# B&R Automation Studio project TD52 (part 107)

#### ERDFCyclic.st - Cyclic code
```iecst
(*********************************************************************************************
AGGR: ERDF task (cyclic)

This code is confidential AND proprietary to the INNIO Company.
It may NOT be used in any form, or reproduced in any manner, without the express
written permission of the INNIO Company.
Copyright, INNIO Company, 2019

Customized modifications: -
------------------------

History:
-------
 V0.1:  Kirchler 02.05.2012: Anwahl Leistungsvorgabe durch ERDF aucb wenn Sollwert über BUS
 							 Signal Aggregat nicht verfügbar wird nicht gesetzt wenn A_ANF fehlt
 V0.2:  Kirchler 17.07.2012: Komplett umgebaut laut vorgabe Clarke; Alle eingänge auf Impuls/flankenauswertung
 							 Leistungsvorgabe und Blindleistungsvorgabe als Reduktion (maximum)
							 RSE Signal implementiert
 V0.3:	Kirchler 13.09.2012: ERDF Schnittstellen aktiv auch im Handbetrieb
 							 Merken der aktuell ausgewählten Cosphi Funktion und nach Beendigung Q0 LIMIT wieder auf alten Wert stellen
							 Vereinfachungen Teil P0- und Q0-Limitierungen
 V0.4:  Kirchler 25.10.2012: Q0 Limitierung Set nur möglich wenn Q0 inaktiv und Reset nur möglich wenn Q0 aktiv.
 							 Verhindert QPF Funktions-Parameter Überschreibungen
							 Wenn Q0_max grösser aktuelle Blindleistung einfach auf alten Cosphi modus zurückschalten
 V0.5:  Adami 07.11.2012: 	 Fehler behoben mit der Netzstörung >50 Sek und der Entkopplung vom netz durch DEIE. Die 2 Funktionen blockierten sich gegenseitig, dadurch
 							 konnte man keine der beiden mehr resetten und die Maschine nicht mehr starten	(außer durch einen Neustart der Diane)
 							 Funktionsänderung der Variablen "DO_NotReady ". Dieser Ausgang dient jetzt als "watchdog", d.h der Ausgang soll immer "1" sein sobald die SPS läuft.
							 Anpassung Blindleistungsreduzierung
 V0.6   Kirchmair 06.02.2014:Erestzen der Variable DI_EVU_3 durch DI_EVU_BLOCK, da sich die Funktion der Variable DI_EVU_3 geändert hat (seit V3.4) und jetzt nicht mehr verwendbar ist.

 V4.00.0 28-04-2014 Maxhera/Waldhart,   implementation OF the module FOR modular software
 V4.03.0 15-03-2016	Perktold,	update FOR 4.3.0.0
 V4.04.0 06-10-2016	Perktold,	update FOR 4.4.0.0 (tiDelayDEIE, IN_GR.tPLim_DEIE.Ai)
		 09.10.2019	lettenb.	div.by zero bugfix, bu01

Instructions FOR use:
--------------------
-
Outstandings:
-------------
*********************************************************************************************)

PROGRAM _CYCLIC

IF Para.bDEIE_Active THEN
(* requirement coupling / decoupling from EU (ERDF), Digital inputs *)
	xSR_MCB_Dcp(SET1 := IN_GR.tMCB_Dcp_SetEUCOn.Di, RESET := IN_GR.tMCB_Dcp_SetEUCOf.Di);
	bMCB_Dcp		 := xSR_MCB_Dcp.Q1;

(* feedback Receive requested Command form machine*)
	IF bMCB_Dcp THEN 						(* True --> hier wird der motor abgefordert *)
		OUT_GR.tMCB_SOn.Do 		:= TRUE;	(* rückmeldung für abforderung *)
		OUT_GR.tERDF_BLOCK.Do 	:= TRUE;   	(* TRUE = abforderung des Motors *)
 	ELSE									(* motor ist wieder freigegeben *)
		OUT_GR.tMCB_SOn.Do		:= FALSE;
		OUT_GR.tERDF_BLOCK.Do 	:= FALSE; 	(* FALSE = keine abforderung des motors durch erdf  *)
	END_IF;

(* =====================================================================*)

(* Freigabe Kopplung ans Netz durch ERDF / Release coupling to the grid by ERDF *)
	xTON_GTE(IN :=  NOT IN_GR.tMnsOk_GTE.Di, PT := Para.tiDelayDEIE);   (* network trouble after X[s]  *)
	xSR_MCB_RelSync(SET1 := IN_GR.tMCB_Rel_Sync.Di, RESET := xTON_GTE.Q);
	bMCB_RelSync := xSR_MCB_RelSync.Q1; (* FALSE = Motor soll blockieren *)

	TP_Msg2888(IN := bMCB_RelSync, PT := T#15s);
	bMsg2888	:= TP_Msg2888.Q;

	IF bMCB_RelSync THEN		(* True --> freigabe für sy erteilt --> keine blockierung *)
		OUT_GR.bOpAlm_ERDF_SY	:= OUT_GR.tMCB_Rel_Sync_SOn.Do := TRUE;	(* rückmeldung und betiebsmeldung abgesetzt *)
	ELSE
		OUT_GR.bOpAlm_ERDF_SY	:= OUT_GR.tMCB_Rel_Sync_SOn.Do := FALSE;
	END_IF;
(* =====================================================================*)

(*  DO: Generator ist eingeschaltet / Generator switch is on *)
	OUT_GR.tGCB_SOn.Do 			:= IN_GR.tGCB_On.Di;
(* =====================================================================*)

(* Fast decoupled by ERDF / Schnelles entkoppeln durch ERDF	*)
(* requirement coupling / decoupling quickly from EU (ERDF), Digital inputs *)
	xSR_MCB_DcpQu(SET1 := IN_GR.tMCB_DcpQu_SetEUCOn.Di, RESET := IN_GR.tMCB_DcpQu_SetEUCOf.Di);
	bMCB_DcpQu	  := xSR_MCB_DcpQu.Q1;

	IF bMCB_DcpQu THEN
		OUT_GR.bOpAlm_DecQu 	:= TRUE;
		OUT_GR.tMCB_EDF_SOn.Do	:= TRUE;
	ELSE
		OUT_GR.bOpAlm_DecQu 	:= FALSE;
		OUT_GR.tMCB_EDF_SOn.Do	:= FALSE;
	END_IF;
(* =====================================================================*)

(*Customers switch for bridging P0 signal / Kundenschalter zur Überbrückung P0 Signal*)
	IF IN_GR.tP0_BLOCK_DEIE.Di THEN
		IN_GR.tPLim_GenC_SetEU.Ai 	:= Para.rP_Set_ExtAI_NormScalMax;
	ELSE
		IN_GR.tPLim_GenC_SetEU.Ai  	:= IN_GR.tP_DEIE.Ai;
	END_IF;

	IF bGCP_PLim AND NOT IN_GR.tP0_BLOCK_DEIE.Di THEN
		OUT_GR.bOpMsg_Plim_ERDF_SOnOf	:= TRUE;
	END_IF;

	IF NOT bGCP_PLim OR  IN_GR.tP0_BLOCK_DEIE.Di THEN
		OUT_GR.bOpMsg_Plim_ERDF_SOnOf	:= FALSE;
	END_IF;

(* powerlimit from ERDF / Leistung reduktion von ERDF *)
	IF  OUT_GR.tPLim_GenC_SOn.Do AND  (IN_GR.tPLim_GenC_SetEU.Ai< (IN_GR.rP_Nom * 0.5)) THEN	(* abforderung des motors sollte die leistungsreduktion < 50% sein *)
		OUT_GR.bOpMsg_Plim_ERDF_ABF_SOnOf	:= TRUE;		(* true = abforderung des Motors *)
	ELSE
		OUT_GR.bOpMsg_Plim_ERDF_ABF_SOnOf 	:= FALSE;
		IN_GR.tPLim_GenC_SetEU.Ai	  		:= LIMIT ((IN_GR.rP_Nom * 0.5), IN_GR.tPLim_GenC_SetEU.Ai,IN_GR.rP_Nom);
		rP_Red_ERDF_Lim			 	  		:= IN_GR.tPLim_GenC_SetEU.Ai / MAX(1, IN_GR.rP_Nom);
	END_IF;
	IF NOT OUT_GR.tPLim_GenC_SOn.Do THEN					(* no powerlimit from ERDF / keine Leistung reduktion über ERDF *)
		rP_Red_ERDF_Lim						:= 1.0; 		(* maximum power / maximale Leistung *)
		OUT_GR.bOpMsg_Plim_ERDF_SOnOf  		:= FALSE;
	END_IF;

(* =====================================================================*)

	IF (bGenC_QLim_ExtRel  OR IN_GR.tP0_BLOCK_DEIE.Di) AND OUT_GR.tQLim_GenC_SOn.Do  THEN
		OUT_GR.bOpMsg_Qlim_ERDF_SOnOf	:= FALSE;
	END_IF

(* =====================================================================*)
// RSE
 (* requirement coupling / decoupling RSE from EU (ERDF), Digital inputs *)
	xSR_RSE(SET1 := IN_GR.tRSE_SetEUCOn.Di, RESET := IN_GR.tRSE_SetEUCOf.Di);
	bRSE	  := xSR_RSE.Q1;

	IF bRSE THEN
		OUT_GR.tRSE_SOn.Do := FALSE;
	ELSE
		OUT_GR.tRSE_SOn.Do := TRUE;
	END_IF;
(* =====================================================================*)

(* =====================================================================*)
	IF OUT_GR.tRSE_SOn.Do THEN
		OUT_GR.bOpMsg_RSE_SOnOf := FALSE;
	END_IF;

	IF NOT OUT_GR.tRSE_SOn.Do THEN
		OUT_GR.bOpMsg_RSE_SOnOf := TRUE;
	END_IF;

// Signal Aggregat verfügbar an ERDF
// Achtung: war früher "Aggregat NICHT Verfügbar", die Logik musste aber umgedreht werden dass der Ausgang 1 ist wenn das Aggregat Verfügbar
// ist, das SPS Label blieb aber gleich damit man den ERDF TAsk einfach austauschen kann ohne die SPS Belegung ändern zu müssen!

	IF IN_GR.tPB2MM.bParaSetupOk THEN
		OUT_GR.tEng_Ready.Do := TRUE;
	ELSE
		OUT_GR.tEng_Ready.Do := FALSE;
	END_IF;
(* =====================================================================*)
(* Output signals interface *)
	OUT_GR.bOpAlm_DecQu;
	OUT_GR.bOpAlm_MSF_P0 		:=	 OUT_GR.tPLim_GenC_SOn.Do AND NOT IN_GR.tP0_BLOCK_DEIE.Di;
	OUT_GR.bOpAlm_ERDF_SY;

	OUT_GR.bOpMsg_Plim_ERDF_SOnOf;
	OUT_GR.bOpMsg_Qlim_ERDF_SOnOf;

	TP_Msg2889(IN := NOT OUT_GR.bOpMsg_Qlim_ERDF_SOnOf, PT := T#15s);
	bMsg2889					:= TP_Msg2889.Q;

	OUT_GR.bOpMsg_RSE_SOnOf;
	OUT_GR.bOpMsg_P0_BLOCK_DEIE_SOnOf := IN_GR.tP0_BLOCK_DEIE.Di;
ELSE
	OUT_GR.tMCB_Rel_Sync_SOn.Do := TRUE;	(* rückmeldung und betiebsmeldung abgesetzt *)
END_IF

END_PROGRAM
```

#### ERDFInit.st - Initialization code
```iecst
(*********************************************************************************************
AGGR: ERDF task (init)

This code is confidential AND proprietary to the INNIO Company.
It may NOT be used in any form, or reproduced in any manner, without the express
written permission of the INNIO Company.
Copyright, INNIO Company, 2019

Customized modifications: -
------------------------

History:
-------

V4.00.0 28-04-2014  Maxhera,   	implementation OF the module FOR modular software
V4.03.0	15.03.2016	Perktold,	update FOR 4.3.0.0

Instructions FOR use:
--------------------
-
Outstandings:
-------------
*********************************************************************************************)
PROGRAM _INIT

;

END_PROGRAM
```

#### ERDF.var - Local variables
```iecst
(********************************************************************
 * COPYRIGHT -- INNIO Company
 ********************************************************************
 * Program: ERDF
 * File: ERDF.var
 * Author: 502297651
 * Created: April 28, 2014
 ********************************************************************
 * Local variables of program ERDF
 ********************************************************************)
VAR
	xSR_MCB_Dcp : SR; (* instance for MCB from DIs*) (* OldName: SR_Plim; Cycle:0; *)
	bMCB_Dcp : BOOL; (* MCB on/off from Digital inputs *) (* OldName: bGCP_Plim; Cycle:0; *)
	xSR_MCB_DcpQu : SR; (* instance for MCB from DIs*) (* OldName: SR_Plim; Cycle:0; *)
	bMCB_DcpQu : BOOL; (* MCB on/off from Digital inputs *) (* OldName: bGCP_Plim; Cycle:0; *)
	xSR_RSE : SR; (* instance for MCB from DIs*) (* OldName: SR_Plim; Cycle:0; *)
	bRSE : BOOL; (* MCB on/off from Digital inputs *) (* OldName: bGCP_Plim; Cycle:0; *)
	xSR_MCB_RelSync : SR; (*instance for MCB_RelSync*) (* OldName: R_TRIG_GCE; Cycle:2; *)
	bMCB_RelSync : BOOL := FALSE;
	xTON_GTE : TON := (0);
	TP_Msg2888 : TP := (0);
	TP_Msg2889 : TP := (0);
END_VAR
```

### Program Logical/Grid/ParGR (IEC, version 4.07.0) - + Parameters Grid Module

- perm_par.st (not readable text: treated as protected, skipped)

#### perm_par.var
```iecst
VAR
	tParaIntern : ParaHandler_typ; (*Connector type to perm_par*)
	tMM2ParaBase_ReadBack : MM2ParaBase_type; (*INTERNAL! V4.06 new readback structure for information from previous tasks*)
	bWriteDataObj : BOOL; (* TRUE=write data object module *)
	bDataObjLenErr : BOOL; (*Error occured in permem: data module size missmatch*)
	bCreateDataObj : BOOL; (* TRUE=create new data object *)
	bWriteOnce : BOOL; (* write permanent memory once *)
	DatObjCreate_01 : DatObjCreate; (* data object create *)
	DatObjInfoBak_02 : DatObjInfo; (* data object info *)
	DatObjDelete_01 : DatObjDelete; (* data object delete *)
	DatObjRead_01 : DatObjRead; (* data object read *)
	DatObjRead_02 : DatObjRead; (* manual initiated data object read *)
	DatObjWrite_01 : DatObjWrite; (* data object write *)
	DatObjDelete_02 : DatObjDelete; (* data object delete *)
	DatObjDelete_11 : DatObjDelete; (*Delete Backup File*)
	DatObjInfo_01 : DatObjInfo; (* data object info *)
	DatObjInfo_02 : DatObjInfo; (* data object info *)
	szModuleName : STRING[35]; (* module name of object *)
	szModuleNameBackup : STRING[35]; (* module name of posiibly created backup object *)
	DatObjCopy_01 : DatObjCopy;
	bCopyDataObj : BOOL;
	TON_WarnDelay : TON;
	TON_WritePMEM : TON; (* delay write permanent memory *)
	ulPMPointer : UDINT; (* adress of actual checksum value *)
	ulChecksum : UDINT; (* parameter checksum value *)
	pm_len : UDINT; (* permanent value lenght *)
	ulChecksumOld : UDINT; (* last vlaue of parameter checksum *)
	ulChkValue : UDINT; (* actual value of parameter pointer *)
	pm_id : UDINT; (* permanent value identifier *)
	pm_p : UDINT; (* permanent value pointer *)
	DatObjInfo_META : DatObjInfo;
	DatObjRead_META : DatObjRead;
	szMetaDataRaw : STRING[2000];
	szMetaData : ARRAY[0..4] OF STRING[35];
	szMetaDataVis : ARRAY[0..3] OF STRING[35];
	ssIndex : INT;
	ssCount : INT;
	ucMetaDataRaw : ARRAY[0..2000] OF USINT;
	ssCount2 : INT;
	szMetaDataFile : STRING[10];
	szText1 : STRING[20];
	pv_adr_IN_XX_tPB2MM : UDINT;
	pv_lng : UDINT;
	pv_lng_IN_XX_tPB2MM : UDINT;
	pv_lng_OUT_XX_tPB2MM : UDINT;
	szText2 : STRING[20];
	pv_adr_OUT_XX_tXX2PB : UDINT;
END_VAR
VAR CONSTANT
	ERR_NOERROR : UINT := 0;
END_VAR
VAR
	usPMWriteCnt : UINT;
	pm_Error : UDINT; (* permanent value error *) (* Deleted: pm : ParaMem_typ; permanent memory tags mathias, 22.8.11*)
	fun_Error : UDINT := 0; (*state > 0 = function error*)
	xLocalParaCheck : ParaCheckFUB; (*local function instance to check parameter values*)
	TON_ParaSetupOk : TON;
	bParaCheckSystemOk : BOOL;
	iDebug_ParaOkChecked : UDINT;
	bRestoreBackupDataObj : BOOL := FALSE;
	bRestoreDataObjContent : BOOL := FALSE;
	pm_id_backup : UDINT;
	pm_p_Backup : UDINT;
	DatObjCopy_02 : DatObjCopy;
	bDeleteBackupDataObj : BOOL := FALSE; (*Command to delete backup data module file on purpose*)
	bDebugPara : ARRAY[0..5] OF BOOL;
	ssIndex2 : INT;
	ssIndex3 : INT;
	ssIndex4 : INT;
	ssIndexVis : INT;
	szText : STRING[40];
	pv_adr_Para : UDINT;
	szParaSnippet : ARRAY[0..5] OF STRING[150];
	szParaIndex : STRING[10];
	slValue : DINT;
	iModuleDLD_ResetCount : INT;
	bDownloadDetected : BOOL;
	bFlagParaStructCopyWorking : BOOL; (*true, if cyclic para copying is active, 1 false cycle at every copy *)
	bStoreInitParaInDataObj : BOOL := FALSE;
	bTestflag : BOOL;
	bReadOutMETA_Once : BOOL;
	tParaCheck_iPvAdress : ARRAY[0..5] OF UDINT;
	tParaCheck_iPvLengt : ARRAY[0..5] OF UDINT;
	tParaCheck_rPvValue : ARRAY[0..5] OF REAL;
	tParaCheck_rRangeMIN : ARRAY[0..5] OF REAL;
	tParaCheck_rRangeMAX : ARRAY[0..5] OF REAL;
	tParaCheck_szPvName : ARRAY[0..5] OF STRING[35];
	ssFormatDetected : INT;
	szMetaDataPart : STRING[150];
	szFullTaskName : STRING[35];
	szFullMetaModuleName : STRING[35];
	debugLen : INT;
	debugSize : INT := 0;
	strcat_adr1 : UDINT;
	strcat_adr2 : UDINT;
	ssIndexTN : INT;
	bAlternate : BOOL;
	n : INT;
	iAlternateChecksum : DINT;
	iAlternateChecksumOld : DINT;
	ulDebugChkValue : ARRAY[0..999] OF UDINT;
	Adr1 : UDINT;
	Adr2 : UDINT;
	usPMWriteCntStepsize : UINT := 1; (*different step sizes to help debug*)
	usPMWriteCntXOR : UINT;
	usPMWriteCntAltSum : UINT;
	ulAdrPM : UDINT;
	usChkValuePM : USINT;
	ulAdrPara : UDINT;
	ulPara_len : UDINT;
	usChkValuePara : USINT;
	iDebugCountPMDifferences : DINT := 0;
	bEngineRunDetected : BOOL; (*detection status bit autocommand 100 /101  for engine run state*)
	ucMetaDataDebugInfoLine : ARRAY[0..24] OF STRING[80];
	ssIndexMand : INT := 0;
	szMetaDataMand : STRING[35];
	iMyErrorInfo_Autoreset : DINT; (*internal autoreset counter*)
	ssIndex_Version : INT; (*internal*)
	ssIndex_BU : INT; (*internal*)
	ssIndex_BU2 : INT; (*internal*)
END_VAR
```

### Program Logical/Grid/MsgGR (IEC, version 4.13.0) - Messages Grid Module

#### MsgGRCyclic.st - Parameters Grid Module
```iecst
(*******************************************************************************
Msg_GR	 			 alarms generation MM_Grid

This code is confidential and proprietary to the INNIO Company.
It may not be used in any form, or reproduced in any manner,
without written permission of the INNIO Company.
Copyright, INNIO Company, 2022

Customized modifications: -
------------------------

History:
-------
V0.01.0	02.11.2011	lettenb.	new
		27.05.2013	lettenb.	reset OUT_xx.txx2AB.bGnlTripx changed
V4.00.0 22-08-2013  Maxhera,    implementation of the module for modular software
		04.03.2014	lettenb.	logger added
		16.06.2015	caks,		clean up
V4.03.0	15-12-2015	Perktold,	Reset fuer alle Warnungen auf TRUE gesetzt + ERDF Meldungen implementiert
								B2812 geaendert fuer HAND Betrieb
V4.03.1	13-06-2016	Gwiggner	Hinzufuegen CustAnaIn[2].Goodqual zu A3385 measuring signal failure P0
V4.04.0	06-10-2016	Perktold	W2799 added changed ERDF to DEIE
V4.04.1	29-03-2017	Gwiggner	add operational messages 2171 and 2172 for frequency control function
V4.05.0 07-12-2017  Farre,		addition op messages from 2940 to 2955 for P and Q functionalities
V4.07.0 28-05-2019	Zuschnig, 	Added A2331, W9261 - W9274 and B3000 B9008 - 9023
V4.10.0	28-09-2020	Zuschnig, 	Changed A2331 logic - NC contact is used
		12.11.2020	lettenb.	2344,2345 added(G99)
V4.11.0	17.01.2022	lettenb.	2812 IN_GR.bEng_Block_EVU added, bugfix
V4.13.0	28.11.2023	Farre,		Enable/disable messages for ILF are added (9093 & 9094)
					Goenczi		2344,2345 Block via BUS added
V4.14.0	17.10.2024	Theobald	Alarm2331 priority changed from 2 to 3 [2024-223]

Instructions for use:
--------------------
1) declare alarm with function block "Alm"
	declare buffert alarm bit bMsg<message number>

2) use template to create a new alarm,
   substitue 0000 by alarm number and make settings:

	xMsg0000.Enable		:=	TRUE;		enable/disable alarm
	xMsg0000.Set		:=	FALSE;		alarm set condition
	xMsg0000.PT			:=	T#0s;		alarm delay time
	xMsg0000.Prio		:=	1;			alarm priority: 1-3 = trip, 4 = warning
	xMsg0000.RiskClass	:=	3;			risk class for remote alarm reset
	xMsg0000.Reset		:=	FALSE;		FALSE: for all standard alarms	prio 1,2,3 and warnings prio 4
										TRUE : for autoreset alarms

	bMsg0000			:=	xMsg0000.Q;	connect buffert alarm bit for VIS and control

3)  expand INIT

3)	include datapoint into OPC configuration for vis

Outstandings:
------------
(*******************************************************************************)
PROGRAM _CYCLIC
	(* reset general trip *)
	OUT_GR.tGR2AB.bGnlTrip1		:=	FALSE;
	OUT_GR.tGR2AB.bGnlTrip2		:=	FALSE;
	OUT_GR.tGR2AB.bGnlTrip3		:=	FALSE;
	OUT_GR.tGR2AB.bGnlWarning	:=	FALSE;
	OUT_GR.tGR2AB.bTriptype1	:=	FALSE;
	OUT_GR.tGR2AB.bTriptype2	:=	FALSE;
	OUT_GR.tGR2AB.bTriptype3	:=	FALSE;

	(*---------------------------------------------------------------------------*)
	(* Trips > AMM *)

	(* A2344 module blocked from grid operator - shutdown *)
	xMsg2344.Enable	   := TRUE;
	xMsg2344.Set	   := IN_GR.tDem_EU_Block2.Di OR IN_GR.bDem_EU_Block2_Bus;
	xMsg2344.PT	   	   := T#0s;
	xMsg2344.Prio 	   := 2;
	xMsg2344.RiskClass := 4;
	xMsg2344.Reset	   := NOT Para.bEU_BlockResetMan; (* autoreset *)
	xMsg2344();
	MM2VIS.bMsg2344    := xMsg2344.Q;
	OUT_GR.tEU_RM_BLOCK2.Do := xMsg2344.Q;

	(* A2345 module blocked from grid operator - demand off *)
	xMsg2345.Enable	   := TRUE;
	xMsg2345.Set	   := IN_GR.tDem_EU_Block3.Di OR IN_GR.bDem_EU_Block3_Bus;
	xMsg2345.PT	   	   := T#0s;
	xMsg2345.Prio 	   := 3;
	xMsg2345.RiskClass := 4;
	xMsg2345.Reset	   := NOT Para.bEU_BlockResetMan; (* autoreset *)
	xMsg2345();
	MM2VIS.bMsg2345    := xMsg2345.Q;
	OUT_GR.tEU_RM_BLOCK3.Do := xMsg2345.Q;

	(* A3384 DEIE fast decoupling *)
	xMsg3384.Enable	   := Para.bDEIE_Active;
	xMsg3384.Set	   := OUT_GR.bOpAlm_DecQu;
	xMsg3384.PT	       := T#0s;
	xMsg3384.Prio 	   := 2;
	xMsg3384.RiskClass := 4;
	xMsg3384();
	MM2VIS.bMsg3384    := xMsg3384.Q;

	(* A3385 measuring signal failure P0 *)
	xMsg3385.Enable	   := Para.bDEIE_Active;
	xMsg3385.Set	   := OUT_GR.bOpAlm_MSF_P0 AND NOT IN_GR.tP_DEIE.GoodQual;
	xMsg3385.PT	       := T#0s;
	xMsg3385.Prio 	   := 3;
	xMsg3385.RiskClass := 4;
	xMsg3385();
	MM2VIS.bMsg3385    := xMsg3385.Q;

	(* A3386 Waiting release for SY DEIE *)
	xMsg3386.Enable	   := Para.bDEIE_Active;
	xMsg3386.Set	   := NOT OUT_GR.bOpAlm_ERDF_SY;
	xMsg3386.Reset	   := IN_GR.tMCB_Rel_Sync.Di;
	xMsg3386.PT	       := T#0s;
	xMsg3386.Prio 	   := 3;
	xMsg3386.RiskClass := 4;
	xMsg3386();
	MM2VIS.bMsg3386    := xMsg3386.Q;

	(* A2331 Surge suppressor has reached critical pressure *)
	IN_GR.tHA2GR.tJunctionBox_GnlAlm.Di := IN_GR.tHA2GR.tJunctionBox_GnlAlm.Di OR NOT IN_GR.tHA2GR.tJunctionBox_GnlAlm.GoodQual;
	xMsg2331.Enable	   := TRUE;
	xMsg2331.Set	   := NOT IN_GR.tHA2GR.tJunctionBox_GnlAlm.Di;
	xMsg2331.Reset	   := FALSE;
	xMsg2331.PT	       := T#0s;
	xMsg2331.Prio 	   := 3;
	xMsg2331.RiskClass := 4;
	xMsg2331();
	MM2VIS.bMsg2331    := xMsg2331.Q;

	(*---------------------------------------------------------------------------*)
	(* Warnings > AMM *)

	(* W3591 - Power limitation by utility operator measuring signal failure *)
	xMsg3591.Enable	   := TRUE;
	xMsg3591.Set	   := bMsg3591;
	xMsg3591.Reset	   := TRUE;
	xMsg3591.PT	       := T#0s;
	xMsg3591.Prio 	   := 4;
	xMsg3591.RiskClass := 4;
	xMsg3591();
	MM2VIS.bMsg3591    := xMsg3591.Q;

	(* W3592 - Power setpoint by utility operator measuring signal failure *)
	xMsg3592.Enable	   := TRUE;
	xMsg3592.Set	   := bMsg3592;
	xMsg3592.Reset	   := TRUE;
	xMsg3592.PT	       := T#0s;
	xMsg3592.Prio 	   := 4;
	xMsg3592.RiskClass := 4;
	xMsg3592();
	MM2VIS.bMsg3592    := xMsg3592.Q;

	(* W3593 - Power factor setpoint by utility operator measuring signal failure *)
	xMsg3593.Enable	   := TRUE;
	xMsg3593.Set	   := bMsg3593;
	xMsg3593.Reset	   := TRUE;
	xMsg3593.PT	       := T#0s;
	xMsg3593.Prio 	   := 4;
	xMsg3593.RiskClass := 4;
	xMsg3593();
	MM2VIS.bMsg3593    := xMsg3593.Q;

	(* W3594 - Reactive power setpoint by utility operator measuring signal failure *)
	xMsg3594.Enable	   := TRUE;
	xMsg3594.Set	   := bMsg3594;
	xMsg3594.Reset	   := TRUE;
	xMsg3594.PT		   := T#0s;
	xMsg3594.Prio 	   := 4;
	xMsg3594.RiskClass := 4;
	xMsg3594();
	MM2VIS.bMsg3594    := xMsg3594.Q;

	(* W3595 - Reactive power limitation by utility operator measuring signal failure *)
	xMsg3595.Enable	   := TRUE;
	xMsg3595.Set	   := bMsg3595;
	xMsg3595.Reset	   := TRUE;
	xMsg3595.PT	   	   := T#0s;
	xMsg3595.Prio 	   := 4;
	xMsg3595.RiskClass := 4;
	xMsg3595();
	MM2VIS.bMsg3595    := xMsg3595.Q;

	(* W3596 - Voltage setpoint by utility operator measuring signal failure *)
	xMsg3596.Enable	   := TRUE;
	xMsg3596.Set	   := bMsg3596;
	xMsg3596.Reset	   := TRUE;
	xMsg3596.PT	   	   := T#0s;
	xMsg3596.Prio 	   := 4;
	xMsg3596.RiskClass := 4;
	xMsg3596();
	MM2VIS.bMsg3596    := xMsg3596.Q;

	(* W2799 - P0 DEIE measuring signal failure *)
	xMsg2799.Enable	   := Para.bDEIE_Active;
	xMsg2799.Set	   := NOT IN_GR.tP_DEIE.GoodQual; (*AND NOT IN_GR.tP0_BLOCK_DEIE.Di;*)
	xMsg2799.Reset	   := TRUE;
	xMsg2799.PT	       := T#0s;
	xMsg2799.Prio 	   := 4;
	xMsg2799.RiskClass := 4;
	xMsg2799();
	MM2VIS.bMsg2799    := xMsg2799.Q;

	(* W9261 - Deadband LFSM-O by utility operator measuring signal failure *)
	xMsg9261.Enable	   := TRUE;
	xMsg9261.Set	   := bMsg9261;
	xMsg9261.Reset	   := TRUE;
	xMsg9261.PT	       := T#0s;
	xMsg9261.Prio 	   := 4;
	xMsg9261.RiskClass := 4;
	xMsg9261();
	MM2VIS.bMsg9261    := xMsg9261.Q;

	(* W9262 - Deadband LFSM-U by utility operator measuring signal failure *)
	xMsg9262.Enable	   := TRUE;
	xMsg9262.Set	   := bMsg9262;
	xMsg9262.Reset	   := TRUE;
	xMsg9262.PT	       := T#0s;
	xMsg9262.Prio 	   := 4;
	xMsg9262.RiskClass := 4;
	xMsg9262();
	MM2VIS.bMsg9262    := xMsg9262.Q;

	(* W9263 - Positive droop LFSM-O by utility operator measuring signal failure *)
	xMsg9263.Enable	   := TRUE;
	xMsg9263.Set	   := bMsg9263;
	xMsg9263.Reset	   := TRUE;
	xMsg9263.PT	       := T#0s;
	xMsg9263.Prio 	   := 4;
	xMsg9263.RiskClass := 4;
	xMsg9263();
	MM2VIS.bMsg9263    := xMsg9263.Q;

	(* W9264 - Negative droop LFSM-U by utility operator measuring signal failure *)
	xMsg9264.Enable	   := TRUE;
	xMsg9264.Set	   := bMsg9264;
	xMsg9264.Reset	   := TRUE;
	xMsg9264.PT	       := T#0s;
	xMsg9264.Prio 	   := 4;
	xMsg9264.RiskClass := 4;
	xMsg9264();
	MM2VIS.bMsg9264    := xMsg9264.Q;

	(* W9265 - Droop FSM-U by utility operator measuring signal failure *)
	xMsg9265.Enable	   := TRUE;
	xMsg9265.Set	   := bMsg9265;
	xMsg9265.Reset	   := TRUE;
	xMsg9265.PT	       := T#0s;
	xMsg9265.Prio 	   := 4;
	xMsg9265.RiskClass := 4;
	xMsg9265();
	MM2VIS.bMsg9265    := xMsg9265.Q;

	(* W9266 - Droop FSM-O by utility operator measuring signal failure *)
	xMsg9266.Enable	   := TRUE;
	xMsg9266.Set	   := bMsg9266;
	xMsg9266.Reset	   := TRUE;
	xMsg9266.PT	       := T#0s;
	xMsg9266.Prio 	   := 4;
	xMsg9266.RiskClass := 4;
	xMsg9266();
	MM2VIS.bMsg9266    := xMsg9266.Q;

	(* W9267 - Dead band FSM-U by utility operator measuring signal failure *)
	xMsg9267.Enable	   := TRUE;
	xMsg9267.Set	   := bMsg9267;
	xMsg9267.Reset	   := TRUE;
	xMsg9267.PT	       := T#0s;
	xMsg9267.Prio 	   := 4;
	xMsg9267.RiskClass := 4;
	xMsg9267();
	MM2VIS.bMsg9267    := xMsg9267.Q;

	(* W9268 - Dead band FSM-O by utility operator measuring signal failure *)
	xMsg9268.Enable	   := TRUE;
	xMsg9268.Set	   := bMsg9268;
	xMsg9268.Reset	   := TRUE;
	xMsg9268.PT	   	   := T#0s;
	xMsg9268.Prio 	   := 4;
	xMsg9268.RiskClass := 4;
	xMsg9268();
	MM2VIS.bMsg9268    := xMsg9268.Q;

	(* W9269 - Positive Margin FSM by utility operator measuring signal failure *)
	xMsg9269.Enable	   := TRUE;
	xMsg9269.Set	   := bMsg9269;
	xMsg9269.Reset	   := TRUE;
	xMsg9269.PT	       := T#0s;
	xMsg9269.Prio 	   := 4;
	xMsg9269.RiskClass := 4;
	xMsg9269();
	MM2VIS.bMsg9269    := xMsg9269.Q;

	(* W9270 - Negative Margin FSM by utility operator measuring signal failure *)
	xMsg9270.Enable	   := TRUE;
	xMsg9270.Set	   := bMsg9270;
	xMsg9270.Reset	   := TRUE;
	xMsg9270.PT	       := T#0s;
	xMsg9270.Prio 	   := 4;
	xMsg9270.RiskClass := 4;
	xMsg9270();
	MM2VIS.bMsg9270    := xMsg9270.Q;

	(* W9271 - U droop by utility operator measuring signal failure *)
	xMsg9271.Enable	   := TRUE;
	xMsg9271.Set	   := bMsg9271;
	xMsg9271.Reset	   := TRUE;
	xMsg9271.PT	       := T#0s;
	xMsg9271.Prio 	   := 4;
	xMsg9271.RiskClass := 4;
	xMsg9271();
	MM2VIS.bMsg9271    := xMsg9271.Q;

	(* W9272 - Ramp rate up by utility operator measuring signal failure *)
	xMsg9272.Enable	   := TRUE;
	xMsg9272.Set	   := bMsg9272;
	xMsg9272.Reset	   := TRUE;
	xMsg9272.PT	       := T#0s;
	xMsg9272.Prio 	   := 4;
	xMsg9272.RiskClass := 4;
	xMsg9272();
	MM2VIS.bMsg9272    := xMsg9272.Q;

	(* W9273 - Ramp rate down by utility operator measuring signal failure *)
	xMsg9273.Enable	   := TRUE;
	xMsg9273.Set	   := bMsg9273;
	xMsg9273.Reset	   := TRUE;
	xMsg9273.PT	   := T#0s;
	xMsg9273.Prio 	   := 4;
	xMsg9273.RiskClass := 4;
	xMsg9273();
	MM2VIS.bMsg9273    := xMsg9273.Q;

	(* W9274 - Reference Frequency FSM/LFSM by utility operator measuring signal failure *)
	xMsg9274.Enable	   := TRUE;
	xMsg9274.Set	   := bMsg9274;
	xMsg9274.Reset	   := TRUE;
	xMsg9274.PT	       := T#0s;
	xMsg9274.Prio 	   := 4;
	xMsg9274.RiskClass := 4;
	xMsg9274();
	MM2VIS.bMsg9274    := xMsg9274.Q;

	(*---------------------------------------------------------------------------*)
	(* operating messages > AMM *)

	(* B2171 - FC response enabled *)
	xMsg2171.Enable		:=	OUT_GR.tGR2CU.bSet_GrC_FSM;
	xMsg2171.Set		:=	OUT_GR.bP_Set_FC_Enable;
	xMsg2171.Reset		:=	TRUE;
	xMsg2171();
	MM2VIS.bMsg2171		:=	xMsg2171.Q;

	(* B2172 - FC response disabled *)
	xMsg2172.Enable		:=	OUT_GR.tGR2CU.bSet_GrC_FSM;
	xMsg2172.Set		:=	NOT OUT_GR.bP_Set_FC_Enable;
	xMsg2172.Reset		:=	TRUE;
	xMsg2172();
	MM2VIS.bMsg2172		:=	xMsg2172.Q;

	(* B2173 - HFR (high frequency response)response enabled *)
	xMsg2173.Enable		:=	Para.bAFC_manual;
	xMsg2173.Set		:=	OUT_GR.bP_Red_POR_Enable;
	xMsg2173.Reset		:=	TRUE;
	xMsg2173();
	MM2VIS.bMsg2173		:=	xMsg2173.Q;

	(* B2174 - HFR response disabled *)
	xMsg2174.Enable		:=	Para.bAFC_manual;
	xMsg2174.Set		:=	NOT OUT_GR.bP_Red_POR_Enable;
	xMsg2174.Reset		:=	TRUE;
	xMsg2174();
	MM2VIS.bMsg2174		:=	xMsg2174.Q;

	(* B2175 - POR response enabled *)
	xMsg2175.Enable		:=	Para.bAFC_manual;
	xMsg2175.Set		:=	OUT_GR.bP_Red_POR_Enable;
	xMsg2175.Reset		:=	TRUE;
	xMsg2175();
	MM2VIS.bMsg2175		:=	xMsg2175.Q;

	(* B2176 - POR response disabled *)
	xMsg2176.Enable		:=	Para.bAFC_manual;
	xMsg2176.Set		:=	NOT OUT_GR.bP_Red_POR_Enable;
	xMsg2176.Reset		:=	TRUE;
	xMsg2176();
	MM2VIS.bMsg2176		:=	xMsg2176.Q;

	(* B2177 - SOR response enabled *)
	xMsg2177.Enable		:=	Para.bAFC_manual;
	xMsg2177.Set		:=	OUT_GR.bP_Red_SOR_Enable;
	xMsg2177.Reset		:=	TRUE;
	xMsg2177();
	MM2VIS.bMsg2177		:=	xMsg2177.Q;

	(* B2178 - SOR response disabled *)
	xMsg2178.Enable		:=	Para.bAFC_manual;
	xMsg2178.Set		:=	NOT OUT_GR.bP_Red_SOR_Enable;
	xMsg2178.Reset		:=	TRUE;
	xMsg2178();
	MM2VIS.bMsg2178		:=	xMsg2178.Q;

	(* B2179 - TOR1 response enabled *)
	xMsg2179.Enable		:=	Para.bAFC_manual;
	xMsg2179.Set		:=	OUT_GR.bP_Red_TOR1_Enable;
	xMsg2179.Reset		:=	TRUE;
	xMsg2179();
	MM2VIS.bMsg2179		:=	xMsg2179.Q;

	(* B2180 - TOR1 response disabled *)
	xMsg2180.Enable		:=	Para.bAFC_manual;
	xMsg2180.Set		:=	NOT OUT_GR.bP_Red_TOR1_Enable;
	xMsg2180.Reset		:=	TRUE;
	xMsg2180();
	MM2VIS.bMsg2180		:=	xMsg2180.Q;

	(* B2181 - TOR2 response enabled *)
	xMsg2181.Enable		:=	Para.bAFC_manual;
	xMsg2181.Set		:=	OUT_GR.bP_Red_TOR2_Enable;
	xMsg2181.Reset		:=	TRUE;
	xMsg2181();
	MM2VIS.bMsg2181		:=	xMsg2181.Q;

	(* B2182 - TOR2 response disabled *)
	xMsg2182.Enable		:=	Para.bAFC_manual;
	xMsg2182.Set		:=	NOT OUT_GR.bP_Red_TOR2_Enable;
	xMsg2182.Reset		:=	TRUE;
	xMsg2182();
	MM2VIS.bMsg2182		:=	xMsg2182.Q;

	(* B2183 - RR response enabled *)
	xMsg2183.Enable		:=	Para.bAFC_manual;
	xMsg2183.Set		:=	OUT_GR.bP_Red_RR_Enable;
	xMsg2183.Reset		:=	TRUE;
	xMsg2183();
	MM2VIS.bMsg2183		:=	xMsg2183.Q;

	(* B2184 - RR response disabled *)
	xMsg2184.Enable		:=	Para.bAFC_manual;
	xMsg2184.Set		:=	NOT OUT_GR.bP_Red_RR_Enable;
	xMsg2184.Reset		:=	TRUE;
	xMsg2184();
	MM2VIS.bMsg2184		:=	xMsg2184.Q;

	(* B2185 - SR response enabled *)
	xMsg2185.Enable		:=	Para.bAFC_manual;
	xMsg2185.Set		:=	OUT_GR.bP_Red_SR_Enable;
	xMsg2185.Reset		:=	TRUE;
	xMsg2185();
	MM2VIS.bMsg2185		:=	xMsg2185.Q;

	(* B2186 - SR response disabled *)
	xMsg2186.Enable		:=	Para.bAFC_manual;
	xMsg2186.Set		:=	NOT OUT_GR.bP_Red_SR_Enable;
	xMsg2186.Reset		:=	TRUE;
	xMsg2186();
	MM2VIS.bMsg2186		:=	xMsg2186.Q;

	(* B2811 power limitation by utility *)
	xMsg2811.Enable		:=	TRUE;
	xMsg2811.Set		:=	IN_GR.PLim_GenC_SetEUPFix1 OR IN_GR.PLim_GenC_SetEUPFix2 OR
							IN_GR.PLim_GenC_SetEUPFix3 OR IN_GR.PLim_GenC_SetEUPFix4 OR
							IN_GR.PLim_GenC_SetEUPFix5;
	xMsg2811.Reset		:=	TRUE;
	xMsg2811();
	MM2VIS.bMsg2811		:=	xMsg2811.Q;

	(* B2812 module blocked by utility *)
	xMsg2812.Enable		:=	TRUE;
	xMsg2812.Set		:=	((IN_GR.tDI_Dem_EU_Block.Di OR IN_GR.bEng_Block_EVU) AND NOT (IN_GR.iIdx_OMSS = 1)) OR bEU_RM_BLOCK_INT OR OUT_GR.tERDF_BLOCK.Do ;
	xMsg2812.Reset		:=	TRUE;
	xMsg2812();
	MM2VIS.bMsg2812		:=	xMsg2812.Q;

	(* B2853 - RMC enabled *)
	xMsg2853.Enable		:=	TRUE;
	xMsg2853.Set		:=	OUT_GR.bP_Red_RMC_Enable;
	xMsg2853.Reset		:=	TRUE;
	xMsg2853();
	MM2VIS.bMsg2853		:=	xMsg2853.Q;

	(* B2854 - RMC disabled *)
	xTP_RMC(IN := EDGENEG(OUT_GR.bP_Red_RMC_Enable), PT := T#10s);

	xMsg2854.Enable		:=	TRUE;
	xMsg2854.Set		:=	xTP_RMC.Q;
	xMsg2854.Reset		:=	TRUE;
	xMsg2854();
	MM2VIS.bMsg2854		:=	xMsg2854.Q;

	(* B2855 - PFC enabled *)
	xMsg2855.Enable		:=	FALSE; (*not in use anymore*)
	xMsg2855.Set		:=	OUT_GR.bP_Red_PFC_Enable;
	xMsg2855.Reset		:=	TRUE;
	xMsg2855();
	MM2VIS.bMsg2855		:=	xMsg2855.Q;

	(* B2856 - PFC disabled *)
	xTP_PFC(IN := EDGENEG(OUT_GR.bP_Red_PFC_Enable), PT := T#10s);

	xMsg2856.Enable		:=	FALSE; (*not in use anymore*)
	xMsg2856.Set		:=	xTP_PFC.Q;
	xMsg2856.Reset		:=	TRUE;
	xMsg2856();
	MM2VIS.bMsg2856		:=	xMsg2856.Q;

	(* B2857 - Power setpoint by utility operator *)
	xMsg2857.Enable		:=	TRUE;
	xMsg2857.Set		:=	OUT_GR.bP_Set_EU_Enable;
	xMsg2857.Reset		:=	TRUE;
	xMsg2857();
	MM2VIS.bMsg2857		:=	xMsg2857.Q;

	(* B2858 - Power factor setpoint by utility operator enabled *)
	xMsg2858.Enable		:=	TRUE;
	xMsg2858.Set		:=	(OUT_GR.iGCQ_Fun_Act = 1);
	xMsg2858.Reset		:=	TRUE;
	xMsg2858();
	MM2VIS.bMsg2858		:=	xMsg2858.Q;

	(* B2859 - Power factor setpoint by utility operator disabled *)
	xTP_PFSet(IN := EDGENEG(OUT_GR.iGCQ_Fun_Act = 1), PT := T#10s);

	xMsg2859.Enable		:=	TRUE;
	xMsg2859.Set		:=	xTP_PFSet.Q;;
	xMsg2859.Reset		:=	TRUE;
	xMsg2859();
	MM2VIS.bMsg2859		:=	xMsg2859.Q;

	(* B2860 - Reactive power setpoint by utility operator enabled *)
	xMsg2860.Enable		:=	TRUE;
	xMsg2860.Set		:=	(OUT_GR.iGCQ_Fun_Act = 6);
	xMsg2860.Reset		:=	TRUE;
	xMsg2860();
	MM2VIS.bMsg2860		:=	xMsg2860.Q;

	(* B2861 - Reactive power setpoint by utility operator disabled *)
	xTP_QSet(IN := EDGENEG(OUT_GR.iGCQ_Fun_Act = 6), PT := T#10s);

	xMsg2861.Enable		:=	TRUE;
	xMsg2861.Set		:=	xTP_QSet.Q;
	xMsg2861.Reset		:=	TRUE;
	xMsg2861();
	MM2VIS.bMsg2861		:=	xMsg2861.Q;

	(* B2862 - Reactive power limitation BY utility operator *)
	xMsg2862.Enable		:=	TRUE;
	xMsg2862.Set		:=	bQLim_Greift;
	xMsg2862.Reset		:=	TRUE;
	xMsg2862();
	MM2VIS.bMsg2862		:=	xMsg2862.Q;

	(* B2863 - Reactive power limitation BY utility operator enabled *)
	xMsg2863.Enable		:=	TRUE;
	xMsg2863.Set		:=	OUT_GR.bQLim_Aktiv ;
	xMsg2863.Reset		:=	TRUE;
	xMsg2863();
	MM2VIS.bMsg2863		:=	xMsg2863.Q;

	(* B2864 - Reactive power limitation BY utility operator disabled *)
	xTP_QLim(IN := EDGENEG(OUT_GR.bQLim_Aktiv), PT := T#10s);

	xMsg2864.Enable		:=	TRUE;
	xMsg2864.Set		:=	xTP_QLim.Q;
	xMsg2864.Reset		:=	TRUE;
	xMsg2864();
	MM2VIS.bMsg2864		:=	xMsg2864.Q;

	(* B2865 - cos phi (P) enabled *)
	xMsg2865.Enable		:=	TRUE;
	xMsg2865.Set		:=	(OUT_GR.iGCQ_Fun_Act = 2);
	xMsg2865.Reset		:=	TRUE;
	xMsg2865();
	MM2VIS.bMsg2865		:=	xMsg2865.Q;

	(* B2866 - cos phi (P) disabled *)
	xTP_PFP(IN := EDGENEG(OUT_GR.iGCQ_Fun_Act = 2), PT := T#10s);

	xMsg2866.Enable		:=	TRUE;
	xMsg2866.Set		:=	xTP_PFP.Q;
	xMsg2866.Reset		:=	TRUE;
	xMsg2866();
	MM2VIS.bMsg2866		:=	xMsg2866.Q;

	(* B2867 - cos phi (U) enabled *)
	xMsg2867.Enable		:=	TRUE;
	xMsg2867.Set		:=	(OUT_GR.iGCQ_Fun_Act = 3);
	xMsg2867.Reset		:=	TRUE;
	xMsg2867();
	MM2VIS.bMsg2867		:=	xMsg2867.Q;

	(* B2868 - cos phi (U) disabled *)
	xTP_PFU(IN := EDGENEG(OUT_GR.iGCQ_Fun_Act = 3), PT := T#10s);

	xMsg2868.Enable		:=	TRUE;
	xMsg2868.Set		:=	xTP_PFU.Q;
	xMsg2868.Reset		:=	TRUE;
	xMsg2868();
	MM2VIS.bMsg2868		:=	xMsg2868.Q;

	(* B2869 - Q(U) enabled *)
	xMsg2869.Enable		:=	TRUE;
	xMsg2869.Set		:=	(OUT_GR.iGCQ_Fun_Act = 4);
	xMsg2869.Reset		:=	TRUE;
	xMsg2869();
	MM2VIS.bMsg2869		:=	xMsg2869.Q;

	(* B2870 - Q(U) disabled *)
	xTP_QU(IN := EDGENEG(OUT_GR.iGCQ_Fun_Act = 4), PT := T#10s);

	xMsg2870.Enable		:=	TRUE;
	xMsg2870.Set		:=	xTP_QU.Q;
	xMsg2870.Reset		:=	TRUE;
	xMsg2870();
	MM2VIS.bMsg2870		:=	xMsg2870.Q;

	(* B2940 - Q customized enabled *)
	xMsg2940.Enable		:=	TRUE;
	xMsg2940.Set		:=	(OUT_GR.iGCQ_Fun_Act = 0) AND (iPrio_Akt = 9);
	xMsg2940.Reset		:=	TRUE;
	xMsg2940();
	MM2VIS.bMsg2940		:=	xMsg2940.Q;

	(* B2941 - Q customized disabled *)
	xTP_QCus(IN := EDGENEG((OUT_GR.iGCQ_Fun_Act = 0) AND (iPrio_Akt = 9)), PT := T#10s);

	xMsg2941.Enable		:=	TRUE;
	xMsg2941.Set		:=	xTP_QCus.Q;
	xMsg2941.Reset		:=	TRUE;
	xMsg2941();
	MM2VIS.bMsg2941		:=	xMsg2941.Q;

	(* B2942 - Voltage control function enabled *)
	xMsg2942.Enable		:=	TRUE;
	xMsg2942.Set		:=	(OUT_GR.iGCQ_Fun_Act = 7);
	xMsg2942.Reset		:=	TRUE;
	xMsg2942();
	MM2VIS.bMsg2942		:=	xMsg2942.Q;

	(* B2943 - Voltage control function  disabled *)
	xTP_UCtrl(IN := EDGENEG(OUT_GR.iGCQ_Fun_Act = 7), PT := T#10s);

	xMsg2943.Enable		:=	TRUE;
	xMsg2943.Set		:=	xTP_UCtrl.Q;
	xMsg2943.Reset		:=	TRUE;
	xMsg2943();
	MM2VIS.bMsg2943		:=	xMsg2943.Q;

	(* B2944 - Q(P) enabled *)
	xMsg2944.Enable		:=	TRUE;
	xMsg2944.Set		:=	(OUT_GR.iGCQ_Fun_Act = 5);
	xMsg2944.Reset		:=	TRUE;
	xMsg2944();
	MM2VIS.bMsg2944		:=	xMsg2944.Q;

	(* B2945 - Q(P) disabled *)
	xTP_QP(IN := EDGENEG(OUT_GR.iGCQ_Fun_Act = 5), PT := T#10s);

	xMsg2945.Enable		:=	TRUE;
	xMsg2945.Set		:=	xTP_QP.Q;
	xMsg2945.Reset		:=	TRUE;
	xMsg2945();
	MM2VIS.bMsg2945		:=	xMsg2945.Q;

	(* B2946 - Function pf-time table enabled *)
	xMsg2946.Enable		:=	TRUE;
	xMsg2946.Set		:=	(OUT_GR.iGCQ_Fun_Act = 8);
	xMsg2946.Reset		:=	TRUE;
	xMsg2946();
	MM2VIS.bMsg2946		:=	xMsg2946.Q;

	(* B2947 - Function pf-time table disabled *)
	xTP_PFP(IN := EDGENEG(OUT_GR.iGCQ_Fun_Act = 8), PT := T#10s);

	xMsg2947.Enable		:=	TRUE;
	xMsg2947.Set		:=	xTP_PFP.Q;
	xMsg2947.Reset		:=	TRUE;
	xMsg2947();
	MM2VIS.bMsg2947		:=	xMsg2947.Q;

	(* B2948 - Test function Q(U), cosphi(U) active *)
	xMsg2948.Enable		:=	TRUE;
	xMsg2948.Set		:=	bSimu_QU_PFU_HMI;
	xMsg2948.Reset		:=	TRUE;
	xMsg2948();
	MM2VIS.bMsg2948		:=	xMsg2948.Q;

	(* B2949 - Q-reduction: Q(U) limitation *)
	xMsg2949.Enable		:=	TRUE;
	xMsg2949.Set		:=	bQ_Lim_QU_Rel;
	xMsg2949.Reset		:=	TRUE;
	xMsg2949();
	MM2VIS.bMsg2949		:=	xMsg2949.Q;

	(* B2950 - LFSM-O activated *)
	xMsg2950.Enable		:=	TRUE;
	xMsg2950.Set		:=	(OUT_GR.bP_Red_PFC_Enable AND Para.bSet_GrC_LFSMO_COn);
	xMsg2950.Reset		:=	TRUE;
	xMsg2950();
	MM2VIS.bMsg2950		:=	xMsg2950.Q;

	(* B2951 - LFSM-O deactivated *)
	xTP_LFSMO(IN := EDGENEG(OUT_GR.bP_Red_PFC_Enable AND Para.bSet_GrC_LFSMO_COn), PT := T#10s);

	xMsg2951.Enable		:=	TRUE;
	xMsg2951.Set		:=	xTP_LFSMO.Q;
	xMsg2951.Reset		:=	TRUE;
	xMsg2951();
	MM2VIS.bMsg2951		:=	xMsg2951.Q;

	(* B2952 - LFSM-U activated *)
	xMsg2952.Enable		:=	TRUE;
	xMsg2952.Set		:=	(OUT_GR.bP_Red_PFC_Enable AND Para.bSet_GrC_LFSMU_COn);
	xMsg2952.Reset		:=	TRUE;
	xMsg2952();
	MM2VIS.bMsg2952		:=	xMsg2952.Q;

	(* B2953 - LFSM-U deactivated *)
	xTP_LFSMU(IN := EDGENEG(OUT_GR.bP_Red_PFC_Enable AND Para.bSet_GrC_LFSMU_COn), PT := T#10s);

	xMsg2953.Enable		:=	TRUE;
	xMsg2953.Set		:=	xTP_LFSMU.Q;
	xMsg2953.Reset		:=	TRUE;
	xMsg2953();
	MM2VIS.bMsg2953		:=	xMsg2953.Q;

	(* B2954 - P(U) activated *)
	xMsg2954.Enable		:=	TRUE;
	xMsg2954.Set		:=	(OUT_GR.bP_Red_PU_Enable);
	xMsg2954.Reset		:=	TRUE;
	xMsg2954();
	MM2VIS.bMsg2954		:=	xMsg2954.Q;

	(* B2955 - P(U) deactivated *)
	xTP_PU(IN := EDGENEG(OUT_GR.bP_Red_PU_Enable), PT := T#10s);

	xMsg2955.Enable		:=	TRUE;
	xMsg2955.Set		:=	xTP_PU.Q;
	xMsg2955.Reset		:=	TRUE;
	xMsg2955();
	MM2VIS.bMsg2955		:=	xMsg2955.Q;

	(* B3000 - Module blocked by Grid module, data structure failure *)
	xMsg3000.Enable		:=	TRUE;
	xMsg3000.Set		:=	OUT_GR.bEng_Bloc_GR;
	xMsg3000.Reset		:=	TRUE;
	xMsg3000();
	MM2VIS.bMsg3000		:=	xMsg3000.Q;

	(* B9008 - LFSMO Droop by utility operator enabled *)
	xMsg9008.Enable		:=	TRUE;
	xMsg9008.Set		:=	bGCP_Droop_GrC_LFSMO_pos OR bBC_Droop_GrC_LFSMO_pos;
	xMsg9008.Reset		:=	TRUE;
	xMsg9008();
	MM2VIS.bMsg9008		:=	xMsg9008.Q;

	(* B9009 - LFSMO Droop by utility operator disabled  *)
	xMsg9009.Enable		:=	TRUE;
	xMsg9009.Set		:=	NOT bGCP_Droop_GrC_LFSMO_pos AND NOT bBC_Droop_GrC_LFSMO_pos;
	xMsg9009.Reset		:=	TRUE;
	xMsg9009();
	MM2VIS.bMsg9009		:=	xMsg9009.Q;

	(* B9010 - LFSMU Droop by utility operator enabled *)
	xMsg9010.Enable		:=	TRUE;
	xMsg9010.Set		:=	bGCP_Droop_GrC_LFSMU_neg OR bBC_Droop_GrC_LFSMU_neg;
	xMsg9010.Reset		:=	TRUE;
	xMsg9010();
	MM2VIS.bMsg9010		:=	xMsg9010.Q;

	(* B9011 - LFSMU Droop by utility operator disabled *)
	xMsg9011.Enable		:=	TRUE;
	xMsg9011.Set		:=	NOT bGCP_Droop_GrC_LFSMU_neg AND NOT bBC_Droop_GrC_LFSMU_neg;
	xMsg9011.Reset		:=	TRUE;
	xMsg9011();
	MM2VIS.bMsg9011		:=	xMsg9011.Q;

	(* B9012 - FSMO Droop by utility operator enabled *)
	xMsg9012.Enable		:=	TRUE;
	xMsg9012.Set		:=	bGCP_Droop_GrC_FSMO OR bBC_Droop_GrC_FSMO;
	xMsg9012.Reset		:=	TRUE;
	xMsg9012();
	MM2VIS.bMsg9012		:=	xMsg9012.Q;

	(* B9013 - FSMO Droop by utility operator disabled *)
	xMsg9013.Enable		:=	TRUE;
	xMsg9013.Set		:=	NOT bGCP_Droop_GrC_FSMO AND NOT bBC_Droop_GrC_FSMO;
	xMsg9013.Reset		:=	TRUE;
	xMsg9013();
	MM2VIS.bMsg9013		:=	xMsg9013.Q;

	(* B9014 - FSMU Droop by utility operator enabled *)
	xMsg9014.Enable		:=	TRUE;
	xMsg9014.Set		:=	bGCP_Droop_GrC_FSMU OR bBC_Droop_GrC_FSMU;
	xMsg9014.Reset		:=	TRUE;
	xMsg9014();
	MM2VIS.bMsg9014		:=	xMsg9014.Q;

	(* B9015 - FSMU Droop by utility operator disabled *)
	xMsg9015.Enable		:=	TRUE;
	xMsg9015.Set		:=	NOT bGCP_Droop_GrC_FSMU AND NOT bBC_Droop_GrC_FSMU;
	xMsg9015.Reset		:=	TRUE;
	xMsg9015();
	MM2VIS.bMsg9015		:=	xMsg9015.Q;

	(* B9016 - FSMO Deadband by utility operator enabled *)
	xMsg9016.Enable		:=	TRUE;
	xMsg9016.Set		:=	bGCP_FSMO_GRC_DB OR bBC_FSMO_GRC_DB;
	xMsg9016.Reset		:=	TRUE;
	xMsg9016();
	MM2VIS.bMsg9016		:=	xMsg9016.Q;

	(* B9017 - FSMO Deadband by utility operator disabled *)
	xMsg9017.Enable		:=	TRUE;
	xMsg9017.Set		:=  NOT	bGCP_FSMO_GRC_DB AND NOT bBC_FSMO_GRC_DB;
	xMsg9017.Reset		:=	TRUE;
	xMsg9017();
	MM2VIS.bMsg9017		:=	xMsg9017.Q;

	(* B9018 - FSMU Deadband by utility operator enabled *)
	xMsg9018.Enable		:=	TRUE;
	xMsg9018.Set		:=	bGCP_FSMU_GRC_DB OR bBC_FSMU_GRC_DB;
	xMsg9018.Reset		:=	TRUE;
	xMsg9018();
	MM2VIS.bMsg9018		:=	xMsg9018.Q;

	(* B9019 - FSMU Deadband by utility operator disabled *)
	xMsg9019.Enable		:=	TRUE;
	xMsg9019.Set		:=  NOT	bGCP_FSMU_GRC_DB AND NOT bBC_FSMU_GRC_DB;
	xMsg9019.Reset		:=	TRUE;
	xMsg9019();
	MM2VIS.bMsg9019		:=	xMsg9019.Q;

	(* B9020 - LFSMO Deadband by utility operator enabled *)
	xMsg9020.Enable		:=	TRUE;
	xMsg9020.Set		:=	bGCP_LFMSO_GRC_DB_pos OR bBC_GCP_LFMSO_GRC_DB_pos;
	xMsg9020.Reset		:=	TRUE;
	xMsg9020();
	MM2VIS.bMsg9020		:=	xMsg9020.Q;

	(* B9021 - LFSMO Deadband by utility operator disabled *)
	xMsg9021.Enable		:=	TRUE;
	xMsg9021.Set		:=	NOT bGCP_LFMSO_GRC_DB_pos AND NOT bBC_GCP_LFMSO_GRC_DB_pos;
	xMsg9021.Reset		:=	TRUE;
	xMsg9021();
	MM2VIS.bMsg9021		:=	xMsg9021.Q;

	(* B9022 - LFSMU Deadband by utility operator enabled *)
	xMsg9022.Enable		:=	TRUE;
	xMsg9022.Set		:=	bGCP_LFMSU_GRC_DB_neg OR bBC_GCP_LFMSU_GRC_DB_neg;
	xMsg9022.Reset		:=	TRUE;
	xMsg9022();
	MM2VIS.bMsg9022		:=	xMsg9022.Q;

	(* B9023 - LFSMU Deadband by utility operator disabled *)
	xMsg9023.Enable		:=	TRUE;
	xMsg9023.Set		:=	NOT bGCP_LFMSU_GRC_DB_neg AND NOT bBC_GCP_LFMSU_GRC_DB_neg;
	xMsg9023.Reset		:=	TRUE;
	xMsg9023();
	MM2VIS.bMsg9023		:=	xMsg9023.Q;

	(* B9093 - ILF enabled *)
	xMsg9093.Enable		:=	TRUE;
	xMsg9093.Set		:=	OUT_GR.bP_Act_ILF_Enable;
	xMsg9093.Reset		:=	TRUE;
	xMsg9093();
	MM2VIS.bMsg9093		:=	xMsg9093.Q;

	(* B9094 - ILF disable *)
	xTP_ILF(IN := EDGENEG(OUT_GR.bP_Act_ILF_Enable), PT := T#10s);

	xMsg9094.Enable		:=	TRUE;
	xMsg9094.Set		:=	xTP_ILF.Q;
	xMsg9094.Reset		:=	TRUE;
	xMsg9094();
	MM2VIS.bMsg9094		:=	xMsg9094.Q;

	IF Para.bDEIE_Active THEN

		xTP_P0(IN := EDGENEG(OUT_GR.bOpMsg_Plim_ERDF_SOnOf), PT := T#15s);

		(* B2886 P0 DEIE activ *)
		MM2VIS.bMsg2886	:= OUT_GR.bOpMsg_Plim_ERDF_SOnOf;

		(* B2887 Q0 DEIE activ *)
		MM2VIS.bMsg2887	:= FALSE; 	(*Standardmeldungen verwerdet*)

		(* B2888 DEIE Release to synchronise *)
		MM2VIS.bMsg2888	:= bMsg2888;

		(* B2889 Q0 not activ *)
		MM2VIS.bMsg2889	:= FALSE;	(*Standardmeldungen verwerdet*)

		(* B2890 RSE activ *)
		MM2VIS.bMsg2890	:= OUT_GR.bOpMsg_RSE_SOnOf;

		(* B2891 P0 not activ *)
		MM2VIS.bMsg2891	:= xTP_P0.Q;

		(* B2892 customer switch on *)
		MM2VIS.bMsg2892	:= OUT_GR.bOpMsg_P0_BLOCK_DEIE_SOnOf;

		(* B2893 customer switch off *)
		MM2VIS.bMsg2893	:= NOT OUT_GR.bOpMsg_P0_BLOCK_DEIE_SOnOf;

	ELSE
		MM2VIS.bMsg2886	:= FALSE;
		MM2VIS.bMsg2887	:= FALSE;
		MM2VIS.bMsg2888	:= FALSE;
		MM2VIS.bMsg2889	:= FALSE;
		MM2VIS.bMsg2890	:= FALSE;
		MM2VIS.bMsg2891	:= FALSE;
		MM2VIS.bMsg2892	:= FALSE;
		MM2VIS.bMsg2893	:= FALSE;
	END_IF;

//	MM2VIS.bMsg2171	:= FALSE;
//	MM2VIS.bMsg2172	:= FALSE;
	MM2VIS.bMsg2173	:= FALSE;
	MM2VIS.bMsg2174	:= FALSE;
	MM2VIS.bMsg2175	:= FALSE;
	MM2VIS.bMsg2176	:= FALSE;
	MM2VIS.bMsg2177	:= FALSE;
	MM2VIS.bMsg2178	:= FALSE;
	MM2VIS.bMsg2179	:= FALSE;
	MM2VIS.bMsg2180	:= FALSE;
	MM2VIS.bMsg2181	:= FALSE;
	MM2VIS.bMsg2182	:= FALSE;
	MM2VIS.bMsg2183	:= FALSE;
	MM2VIS.bMsg2184	:= FALSE;
	MM2VIS.bMsg2185	:= FALSE;
	MM2VIS.bMsg2186	:= FALSE;

	(* B template
	xMsg.Enable		:=	TRUE;
	xMsg.Set		:=	bBool;
	xMsg.Reset		:=	TRUE;
	xMsg();
	MM2VIS.bMsg		:=	xMsg.Q;	*)

	(*--------------------------------------------------------------------------*)
	(* general alarms for further module operations *)
	bGnlTrip1	:= OUT_GR.tGR2AB.bGnlTrip1   OR IN_GR.tAB2GR.bGnlTrip1;
	bGnlTrip2	:= OUT_GR.tGR2AB.bGnlTrip2   OR IN_GR.tAB2GR.bGnlTrip2;
	bGnlTrip3	:= OUT_GR.tGR2AB.bGnlTrip3   OR IN_GR.tAB2GR.bGnlTrip3;
	bGnlWarning	:= OUT_GR.tGR2AB.bGnlWarning OR IN_GR.tAB2GR.bGnlWarning;

	bGnlTrip	:=	bGnlTrip1 OR bGnlTrip2 OR bGnlTrip3;

	(*******************************************************************************)
END_PROGRAM
```

#### MsgGRInit.st - Parameters Grid Module init
```iecst
(*******************************************************************************
Msg_VE	 			 alarms generation MM_ventilation

This code is confidential and proprietary to the INNIO Company.
It may not be used in any form, or reproduced in any manner,
without written permission of the INNIO Company.
Copyright, INNIO Company, 2019

Customized modifications: -
------------------------

History:
-------
V0.00.0	29.07.2011	lettenb.	new
V4.00.0 22-08-2013  Maxhera,   	implementation of the module for modular software
V4.03.0	15-12-2015	Perktold,	Reset für alle Warnungen auf TRUE gesetzt + ERDF Meldungen implementiert
V4.04.0	06-10-2016	Perktold	added W2799

Instructions for use:
--------------------
1) declare alarm with function block "Msg"

2) use template to create a new alarm, substitue 0000 by message number:

	xMsg0000.Num		:=	0000;					alarm number
	xMsg0000.AmmSysAdr	:=  iAdrAmmBase2MM;			do not change
	xMsg0000.AmmOutAdr	:=  iAdrMM2AmmBase;			do not change

3) 	set alarm number

Outstandings:
------------
(*******************************************************************************)
PROGRAM _INIT

	iAdrAmmBase2MM		:=  ADR(IN_GR.tAB2GR);
	iAdrMM2AmmBase		:=  ADR(OUT_GR.tGR2AB);

	xMsg2171.Num		:= 	2171;
	xMsg2171.AmmInAdr	:=  iAdrAmmBase2MM;
	xMsg2171.AmmOutAdr	:=  iAdrMM2AmmBase;

	xMsg2172.Num		:= 	2172;
	xMsg2172.AmmInAdr	:=  iAdrAmmBase2MM;
	xMsg2172.AmmOutAdr	:=  iAdrMM2AmmBase;

	xMsg2173.Num		:= 	2173;
	xMsg2173.AmmInAdr	:=  iAdrAmmBase2MM;
	xMsg2173.AmmOutAdr	:=  iAdrMM2AmmBase;

	xMsg2174.Num		:= 	2174;
	xMsg2174.AmmInAdr	:=  iAdrAmmBase2MM;
	xMsg2174.AmmOutAdr	:=  iAdrMM2AmmBase;

	xMsg2175.Num		:=	2175;
	xMsg2175.AmmInAdr	:=  iAdrAmmBase2MM;
	xMsg2175.AmmOutAdr	:=  iAdrMM2AmmBase;

	xMsg2176.Num		:= 	2176;
	xMsg2176.AmmInAdr	:=  iAdrAmmBase2MM;
	xMsg2176.AmmOutAdr	:=  iAdrMM2AmmBase;

	xMsg2177.Num		:= 	2177;
	xMsg2177.AmmInAdr	:=  iAdrAmmBase2MM;
	xMsg2177.AmmOutAdr	:=  iAdrMM2AmmBase;

	xMsg2178.Num		:= 	2178;
	xMsg2178.AmmInAdr	:=  iAdrAmmBase2MM;
	xMsg2178.AmmOutAdr	:=  iAdrMM2AmmBase;

	xMsg2179.Num		:= 	2179;
	xMsg2179.AmmInAdr	:=  iAdrAmmBase2MM;
	xMsg2179.AmmOutAdr	:=  iAdrMM2AmmBase;

	xMsg2180.Num		:= 	2180;
	xMsg2180.AmmInAdr	:=  iAdrAmmBase2MM;
	xMsg2180.AmmOutAdr	:=  iAdrMM2AmmBase;

	xMsg2181.Num		:= 	2181;
	xMsg2181.AmmInAdr	:=  iAdrAmmBase2MM;
	xMsg2181.AmmOutAdr	:=  iAdrMM2AmmBase;

	xMsg2182.Num		:= 	2182;
	xMsg2182.AmmInAdr	:=  iAdrAmmBase2MM;
	xMsg2182.AmmOutAdr	:=  iAdrMM2AmmBase;

	xMsg2183.Num		:= 	2183;
	xMsg2183.AmmInAdr	:=  iAdrAmmBase2MM;
	xMsg2183.AmmOutAdr	:=  iAdrMM2AmmBase;

	xMsg2184.Num		:=	2184;
	xMsg2184.AmmInAdr	:=  iAdrAmmBase2MM;
	xMsg2184.AmmOutAdr	:=  iAdrMM2AmmBase;

	xMsg2185.Num		:= 	2185;
	xMsg2185.AmmInAdr	:=  iAdrAmmBase2MM;
	xMsg2185.AmmOutAdr	:=  iAdrMM2AmmBase;

	xMsg2186.Num		:= 	2186;
	xMsg2186.AmmInAdr	:=  iAdrAmmBase2MM;
	xMsg2186.AmmOutAdr	:=  iAdrMM2AmmBase;

	xMsg2344.Num		:= 	2344;
	xMsg2344.AmmInAdr	:=  iAdrAmmBase2MM;
	xMsg2344.AmmOutAdr	:=  iAdrMM2AmmBase;

	xMsg2345.Num		:= 	2345;
	xMsg2345.AmmInAdr	:=  iAdrAmmBase2MM;
	xMsg2345.AmmOutAdr	:=  iAdrMM2AmmBase;

	xMsg2811.Num		:= 	2811;
	xMsg2811.AmmInAdr	:=  iAdrAmmBase2MM;
	xMsg2811.AmmOutAdr	:=  iAdrMM2AmmBase;

	xMsg2812.Num		:= 	2812;
	xMsg2812.AmmInAdr	:=  iAdrAmmBase2MM;
	xMsg2812.AmmOutAdr	:=  iAdrMM2AmmBase;

	xMsg2853.Num		:= 	2853;
	xMsg2853.AmmInAdr	:=  iAdrAmmBase2MM;
	xMsg2853.AmmOutAdr	:=  iAdrMM2AmmBase;

	xMsg2854.Num		:= 	2854;
	xMsg2854.AmmInAdr	:=  iAdrAmmBase2MM;
	xMsg2854.AmmOutAdr	:=  iAdrMM2AmmBase;

	xMsg2855.Num		:= 	2855;
	xMsg2855.AmmInAdr	:=  iAdrAmmBase2MM;
	xMsg2855.AmmOutAdr	:=  iAdrMM2AmmBase;

	xMsg2856.Num		:= 	2856;
	xMsg2856.AmmInAdr	:=  iAdrAmmBase2MM;
	xMsg2856.AmmOutAdr	:=  iAdrMM2AmmBase;

	xMsg2857.Num		:= 	2857;
	xMsg2857.AmmInAdr	:=  iAdrAmmBase2MM;
	xMsg2857.AmmOutAdr	:=  iAdrMM2AmmBase;

	xMsg2858.Num		:= 	2858;
	xMsg2858.AmmInAdr	:=  iAdrAmmBase2MM;
	xMsg2858.AmmOutAdr	:=  iAdrMM2AmmBase;

	xMsg2859.Num		:= 	2859;
	xMsg2859.AmmInAdr	:=  iAdrAmmBase2MM;
	xMsg2859.AmmOutAdr	:=  iAdrMM2AmmBase;

	xMsg2860.Num		:= 	2860;
	xMsg2860.AmmInAdr	:=  iAdrAmmBase2MM;
	xMsg2860.AmmOutAdr	:=  iAdrMM2AmmBase;

	xMsg2861.Num		:= 	2861;
	xMsg2861.AmmInAdr	:=  iAdrAmmBase2MM;
	xMsg2861.AmmOutAdr	:=  iAdrMM2AmmBase;

	xMsg2862.Num		:= 	2862;
	xMsg2862.AmmInAdr	:=  iAdrAmmBase2MM;
	xMsg2862.AmmOutAdr	:=  iAdrMM2AmmBase;

	xMsg2863.Num		:= 	2863;
	xMsg2863.AmmInAdr	:=  iAdrAmmBase2MM;
	xMsg2863.AmmOutAdr	:=  iAdrMM2AmmBase;

	xMsg2864.Num		:= 	2864;
	xMsg2864.AmmInAdr	:=  iAdrAmmBase2MM;
	xMsg2864.AmmOutAdr	:=  iAdrMM2AmmBase;

	xMsg2865.Num		:=  2865;
	xMsg2865.AmmInAdr	:=  iAdrAmmBase2MM;
	xMsg2865.AmmOutAdr	:=  iAdrMM2AmmBase;

	xMsg2866.Num		:=  2866;
	xMsg2866.AmmInAdr	:=  iAdrAmmBase2MM;
	xMsg2866.AmmOutAdr	:=  iAdrMM2AmmBase;

	xMsg2867.Num		:=  2867;
	xMsg2867.AmmInAdr	:=  iAdrAmmBase2MM;
	xMsg2867.AmmOutAdr	:=  iAdrMM2AmmBase;

	xMsg2868.Num		:=  2868;
	xMsg2868.AmmInAdr	:=  iAdrAmmBase2MM;
	xMsg2868.AmmOutAdr	:=  iAdrMM2AmmBase;

	xMsg2869.Num		:=  2869;
	xMsg2869.AmmInAdr	:=  iAdrAmmBase2MM;
	xMsg2869.AmmOutAdr	:=  iAdrMM2AmmBase;

	xMsg2870.Num		:=  2870;
	xMsg2870.AmmInAdr	:=  iAdrAmmBase2MM;
	xMsg2870.AmmOutAdr	:=  iAdrMM2AmmBase;

	xMsg2870.Num		:=  2870;
	xMsg2870.AmmInAdr	:=  iAdrAmmBase2MM;
	xMsg2870.AmmOutAdr	:=  iAdrMM2AmmBase;

	xMsg3384.Num		:= 	3384;
	xMsg3384.AmmInAdr	:=  iAdrAmmBase2MM;
	xMsg3384.AmmOutAdr	:=  iAdrMM2AmmBase;

	xMsg3385.Num		:= 	3385;
	xMsg3385.AmmInAdr	:=  iAdrAmmBase2MM;
	xMsg3385.AmmOutAdr	:=  iAdrMM2AmmBase;

	xMsg3386.Num		:= 	3386;
	xMsg3386.AmmInAdr	:=  iAdrAmmBase2MM;
	xMsg3386.AmmOutAdr	:=  iAdrMM2AmmBase;

	xMsg3591.Num		:=  3591;
	xMsg3591.AmmInAdr	:=  iAdrAmmBase2MM;
	xMsg3591.AmmOutAdr	:=  iAdrMM2AmmBase;

	xMsg3592.Num		:=  3592;
	xMsg3592.AmmInAdr	:=  iAdrAmmBase2MM;
	xMsg3592.AmmOutAdr	:=  iAdrMM2AmmBase;

	xMsg3593.Num		:=  3593;
	xMsg3593.AmmInAdr	:=  iAdrAmmBase2MM;
	xMsg3593.AmmOutAdr	:=  iAdrMM2AmmBase;

	xMsg3594.Num		:=  3594;
	xMsg3594.AmmInAdr	:=  iAdrAmmBase2MM;
	xMsg3594.AmmOutAdr	:=  iAdrMM2AmmBase;

	xMsg3595.Num		:=  3595;
	xMsg3595.AmmInAdr	:=  iAdrAmmBase2MM;
	xMsg3595.AmmOutAdr	:=  iAdrMM2AmmBase;

	xMsg3596.Num		:=  3596;
	xMsg3596.AmmInAdr	:=  iAdrAmmBase2MM;
	xMsg3596.AmmOutAdr	:=  iAdrMM2AmmBase;

	xMsg2799.Num		:=  2799;
	xMsg2799.AmmInAdr	:=  iAdrAmmBase2MM;
	xMsg2799.AmmOutAdr	:=  iAdrMM2AmmBase;

	xMsg2940.Num		:=  2940;
	xMsg2940.AmmInAdr	:=  iAdrAmmBase2MM;
	xMsg2940.AmmOutAdr	:=  iAdrMM2AmmBase;

	xMsg2941.Num		:=  2941;
	xMsg2941.AmmInAdr	:=  iAdrAmmBase2MM;
	xMsg2941.AmmOutAdr	:=  iAdrMM2AmmBase;

	xMsg2942.Num		:=  2942;
	xMsg2942.AmmInAdr	:=  iAdrAmmBase2MM;
	xMsg2942.AmmOutAdr	:=  iAdrMM2AmmBase;

	xMsg2943.Num		:=  2943;
	xMsg2943.AmmInAdr	:=  iAdrAmmBase2MM;
	xMsg2943.AmmOutAdr	:=  iAdrMM2AmmBase;

	xMsg2944.Num		:=  2944;
	xMsg2944.AmmInAdr	:=  iAdrAmmBase2MM;
	xMsg2944.AmmOutAdr	:=  iAdrMM2AmmBase;

	xMsg2945.Num		:=  2945;
	xMsg2945.AmmInAdr	:=  iAdrAmmBase2MM;
	xMsg2945.AmmOutAdr	:=  iAdrMM2AmmBase;

	xMsg2946.Num		:=  2946;
	xMsg2946.AmmInAdr	:=  iAdrAmmBase2MM;
	xMsg2946.AmmOutAdr	:=  iAdrMM2AmmBase;

	xMsg2947.Num		:=  2947;
	xMsg2947.AmmInAdr	:=  iAdrAmmBase2MM;
	xMsg2947.AmmOutAdr	:=  iAdrMM2AmmBase;

	xMsg2948.Num		:=  2948;
	xMsg2948.AmmInAdr	:=  iAdrAmmBase2MM;
	xMsg2948.AmmOutAdr	:=  iAdrMM2AmmBase;

	xMsg2949.Num		:=  2949;
	xMsg2949.AmmInAdr	:=  iAdrAmmBase2MM;
	xMsg2949.AmmOutAdr	:=  iAdrMM2AmmBase;

	xMsg2950.Num		:=  2950;
	xMsg2950.AmmInAdr	:=  iAdrAmmBase2MM;
	xMsg2950.AmmOutAdr	:=  iAdrMM2AmmBase;

	xMsg2951.Num		:=  2951;
	xMsg2951.AmmInAdr	:=  iAdrAmmBase2MM;
	xMsg2951.AmmOutAdr	:=  iAdrMM2AmmBase;

	xMsg2952.Num		:=  2952;
	xMsg2952.AmmInAdr	:=  iAdrAmmBase2MM;
	xMsg2952.AmmOutAdr	:=  iAdrMM2AmmBase;

	xMsg2953.Num		:=  2953;
	xMsg2953.AmmInAdr	:=  iAdrAmmBase2MM;
	xMsg2953.AmmOutAdr	:=  iAdrMM2AmmBase;

	xMsg2954.Num		:=  2954;
	xMsg2954.AmmInAdr	:=  iAdrAmmBase2MM;
	xMsg2954.AmmOutAdr	:=  iAdrMM2AmmBase;

	xMsg2955.Num		:=  2955;
	xMsg2955.AmmInAdr	:=  iAdrAmmBase2MM;
	xMsg2955.AmmOutAdr	:=  iAdrMM2AmmBase;

	xMsg2331.Num		:=  2331;
	xMsg2331.AmmInAdr	:=  iAdrAmmBase2MM;
	xMsg2331.AmmOutAdr	:=  iAdrMM2AmmBase;

	xMsg3000.Num		:=	3000;
	xMsg3000.AmmInAdr	:=	iAdrAmmBase2MM;
	xMsg3000.AmmOutAdr	:=	iAdrMM2AmmBase;

	xMsg9261.Num		:=  9261;
	xMsg9261.AmmInAdr	:=  iAdrAmmBase2MM;
	xMsg9261.AmmOutAdr	:=  iAdrMM2AmmBase;

	xMsg9262.Num		:=  9262;
	xMsg9262.AmmInAdr	:=  iAdrAmmBase2MM;
	xMsg9262.AmmOutAdr	:=  iAdrMM2AmmBase;

	xMsg9263.Num		:=  9263;
	xMsg9263.AmmInAdr	:=  iAdrAmmBase2MM;
	xMsg9263.AmmOutAdr	:=  iAdrMM2AmmBase;

	xMsg9264.Num		:=  9264;
	xMsg9264.AmmInAdr	:=  iAdrAmmBase2MM;
	xMsg9264.AmmOutAdr	:=  iAdrMM2AmmBase;

	xMsg9265.Num		:=  9265;
	xMsg9265.AmmInAdr	:=  iAdrAmmBase2MM;
	xMsg9265.AmmOutAdr	:=  iAdrMM2AmmBase;

	xMsg9266.Num		:=  9266;
	xMsg9266.AmmInAdr	:=  iAdrAmmBase2MM;
	xMsg9266.AmmOutAdr	:=  iAdrMM2AmmBase;

	xMsg9267.Num		:=  9267;
	xMsg9267.AmmInAdr	:=  iAdrAmmBase2MM;
	xMsg9267.AmmOutAdr	:=  iAdrMM2AmmBase;

	xMsg9268.Num		:=  9268;
	xMsg9268.AmmInAdr	:=  iAdrAmmBase2MM;
	xMsg9268.AmmOutAdr	:=  iAdrMM2AmmBase;

	xMsg9269.Num		:=  9269;
	xMsg9269.AmmInAdr	:=  iAdrAmmBase2MM;
	xMsg9269.AmmOutAdr	:=  iAdrMM2AmmBase;

	xMsg9270.Num		:=  9270;
	xMsg9270.AmmInAdr	:=  iAdrAmmBase2MM;
	xMsg9270.AmmOutAdr	:=  iAdrMM2AmmBase;

	xMsg9271.Num		:=  9271;
	xMsg9271.AmmInAdr	:=  iAdrAmmBase2MM;
	xMsg9271.AmmOutAdr	:=  iAdrMM2AmmBase;

	xMsg9272.Num		:=  9272;
	xMsg9272.AmmInAdr	:=  iAdrAmmBase2MM;
	xMsg9272.AmmOutAdr	:=  iAdrMM2AmmBase;

	xMsg9273.Num		:=  9273;
	xMsg9273.AmmInAdr	:=  iAdrAmmBase2MM;
	xMsg9273.AmmOutAdr	:=  iAdrMM2AmmBase;

	xMsg9274.Num		:=  9274;
	xMsg9274.AmmInAdr	:=  iAdrAmmBase2MM;
	xMsg9274.AmmOutAdr	:=  iAdrMM2AmmBase;

	xMsg9008.Num		:=  9008;
	xMsg9008.AmmInAdr	:=  iAdrAmmBase2MM;
	xMsg9008.AmmOutAdr	:=  iAdrMM2AmmBase;

	xMsg9009.Num		:=	9009;
	xMsg9009.AmmInAdr	:=	iAdrAmmBase2MM;
	xMsg9009.AmmOutAdr	:=	iAdrMM2AmmBase;

	xMsg9010.Num		:=	9010;
	xMsg9010.AmmInAdr	:=	iAdrAmmBase2MM;
	xMsg9010.AmmOutAdr	:=	iAdrMM2AmmBase;

	xMsg9011.Num		:=	9011;
	xMsg9011.AmmInAdr	:=	iAdrAmmBase2MM;
	xMsg9011.AmmOutAdr	:=	iAdrMM2AmmBase;

	xMsg9012.Num		:=	9012;
	xMsg9012.AmmInAdr	:=	iAdrAmmBase2MM;
	xMsg9012.AmmOutAdr	:=	iAdrMM2AmmBase;

	xMsg9013.Num		:=	9013;
	xMsg9013.AmmInAdr	:=	iAdrAmmBase2MM;
	xMsg9013.AmmOutAdr	:=	iAdrMM2AmmBase;

	xMsg9014.Num		:=	9014;
	xMsg9014.AmmInAdr	:=	iAdrAmmBase2MM;
	xMsg9014.AmmOutAdr	:=	iAdrMM2AmmBase;

	xMsg9015.Num		:=	9015;
	xMsg9015.AmmInAdr	:=	iAdrAmmBase2MM;
	xMsg9015.AmmOutAdr	:=	iAdrMM2AmmBase;

	xMsg9016.Num		:=	9016;
	xMsg9016.AmmInAdr	:=	iAdrAmmBase2MM;
	xMsg9016.AmmOutAdr	:=	iAdrMM2AmmBase;

	xMsg9017.Num		:=	9017;
	xMsg9017.AmmInAdr	:=	iAdrAmmBase2MM;
	xMsg9017.AmmOutAdr	:=	iAdrMM2AmmBase;

	xMsg9018.Num		:=	9018;
	xMsg9018.AmmInAdr	:=	iAdrAmmBase2MM;
	xMsg9018.AmmOutAdr	:=	iAdrMM2AmmBase;

	xMsg9019.Num		:=	9019;
	xMsg9019.AmmInAdr	:=	iAdrAmmBase2MM;
	xMsg9019.AmmOutAdr	:=	iAdrMM2AmmBase;

	xMsg9020.Num		:=	9020;
	xMsg9020.AmmInAdr	:=	iAdrAmmBase2MM;
	xMsg9020.AmmOutAdr	:=	iAdrMM2AmmBase;

	xMsg9021.Num		:=	9021;
	xMsg9021.AmmInAdr	:=	iAdrAmmBase2MM;
	xMsg9021.AmmOutAdr	:=	iAdrMM2AmmBase;

	xMsg9022.Num		:=	9022;
	xMsg9022.AmmInAdr	:=	iAdrAmmBase2MM;
	xMsg9022.AmmOutAdr	:=	iAdrMM2AmmBase;

	xMsg9023.Num		:=	9023;
	xMsg9023.AmmInAdr	:=	iAdrAmmBase2MM;
	xMsg9023.AmmOutAdr	:=	iAdrMM2AmmBase;

	xMsg9093.Num		:=	9093;
	xMsg9093.AmmInAdr	:=	iAdrAmmBase2MM;
	xMsg9093.AmmOutAdr	:=	iAdrMM2AmmBase;

	xMsg9094.Num		:=	9094;
	xMsg9094.AmmInAdr	:=	iAdrAmmBase2MM;
	xMsg9094.AmmOutAdr	:=	iAdrMM2AmmBase;

END_PROGRAM
```

#### MsgGR.var
```iecst
VAR
	iAdrMM2AmmBase : UDINT;
	iAdrAmmBase2MM : UDINT;
	xMsg2811 : Msg; (* B2811 power limitation by utility *)
	xMsg2812 : Msg; (* B2812 module blocked by utility *)
	xMsg2853 : Msg; (* B2853 -  instance of AmBase Library function Msg*)
	xMsg2854 : Msg; (* B2854 -  instance of AmBase Library function Msg*)
	xMsg2855 : Msg; (* B2855 -  instance of AmBase Library function Msg*)
	xMsg2856 : Msg; (* B2856 -  instance of AmBase Library function Msg*)
	xMsg2857 : Msg; (* B2857 -  instance of AmBase Library function Msg*)
	xMsg2858 : Msg; (* B2858 -  instance of AmBase Library function Msg*)
	xMsg2859 : Msg; (* B2859 -  instance of AmBase Library function Msg*)
	xMsg2860 : Msg; (* B2860 -  instance of AmBase Library function Msg*)
	xMsg2861 : Msg; (* B2861 -  instance of AmBase Library function Msg*)
	xMsg2862 : Msg; (* B2862 -  instance of AmBase Library function Msg*)
	xMsg2863 : Msg; (* B2863 -  instance of AmBase Library function Msg*)
	xMsg2864 : Msg; (* B2864 -  instance of AmBase Library function Msg*)
	xMsg2865 : Msg; (* B2865 -  instance of AmBase Library function Msg*)
	xMsg2866 : Msg; (* B2866 -  instance of AmBase Library function Msg*)
	xMsg2867 : Msg; (* B2867 -  instance of AmBase Library function Msg*)
	xMsg2868 : Msg; (* B2868 -  instance of AmBase Library function Msg*)
	xMsg2869 : Msg; (* B2869 -  instance of AmBase Library function Msg*)
	xMsg3384 : Msg; (* A3384 - instance of AmBase Library function Msg*)
	xMsg3385 : Msg; (* A3385 - instance of AmBase Library function Msg*)
	xMsg3386 : Msg; (* A3386 - instance of AmBase Library function Msg *)
	xMsg2870 : Msg; (* B2870 -  instance of AmBase Library function Msg*)
	xMsg3591 : Msg; (* W2891 -  instance of AmBase Library function Msg*)
	xMsg3592 : Msg; (* W2892 -  instance of AmBase Library function Msg*)
	xMsg3593 : Msg; (* W2893 -  instance of AmBase Library function Msg*)
	xMsg3594 : Msg; (* W2894 -  instance of AmBase Library function Msg*)
	xMsg2799 : Msg; (* W2799 -  P0 DEIE measuring signal failure*)
	xMsg3595 : Msg; (* W2895 -  instance of AmBase Library function Msg*)
	xMsg3596 : Msg; (* W2896 -  instance of AmBase Library function Msg*)
	xMsg2331 : Msg; (* A2331 -  instance of AmBase Library function Msg*)
	xMsg3000 : Msg; (* W3000 -  instance of AmBase Library function Msg*)
	xMsg9261 : Msg; (* W9261 -  instance of AmBase Library function Msg*)
	xMsg9262 : Msg; (* W9262 -  instance of AmBase Library function Msg*)
	xMsg9263 : Msg; (* W9263 -  instance of AmBase Library function Msg*)
	xMsg9264 : Msg; (* W9264 -  instance of AmBase Library function Msg*)
	xMsg9265 : Msg; (* W9265 -  instance of AmBase Library function Msg*)
	xMsg9266 : Msg; (* W9266 -  instance of AmBase Library function Msg*)
	xMsg9267 : Msg; (* W9267 -  instance of AmBase Library function Msg*)
	xMsg9268 : Msg; (* W9268 -  instance of AmBase Library function Msg*)
	xMsg9269 : Msg; (* W9269 -  instance of AmBase Library function Msg*)
	xMsg9270 : Msg; (* W9270 -  instance of AmBase Library function Msg*)
	xMsg9271 : Msg; (* W9271 -  instance of AmBase Library function Msg*)
	xMsg9272 : Msg; (* W9272 -  instance of AmBase Library function Msg*)
	xMsg9273 : Msg; (* W9273 -  instance of AmBase Library function Msg*)
	xMsg9274 : Msg; (* W9274 -  instance of AmBase Library function Msg*)
	xTP_RMC : TP; (* 0 implements a pulse generator*) (* OldName: TP_RMC; Cycle:0; *)
	xTP_PFC : TP; (* implements a pulse generator*) (* OldName: TP_PFC; Cycle:0; *)
	xTP_PFSet : TP := (0);
	xTP_QSet : TP := (0);
	xTP_PFP : TP := (0);
	xTP_PFU : TP := (0);
	xTP_QLim : TP := (0);
	xTP_QCus : TP := (0);
	xTP_UCtrl : TP := (0);
	xTP_QU : TP := (0);
	xTP_LFSMO : TP := (0);
	xTP_LFSMU : TP := (0);
	xTP_ILF : TP := (0);
	xTP_QP : TP := (0);
	xTP_PU : TP := (0);
	xMsg2171 : Msg;
	xMsg2172 : Msg;
	xMsg2173 : Msg;
	xMsg2174 : Msg;
	xMsg2175 : Msg;
	xMsg2176 : Msg;
	xMsg2177 : Msg;
	xMsg2178 : Msg;
	xMsg2179 : Msg;
	xMsg2180 : Msg;
	xMsg2181 : Msg;
	xMsg2182 : Msg;
	xMsg2183 : Msg;
	xMsg2184 : Msg;
	xMsg2185 : Msg;
	xMsg2186 : Msg;
	xTP_P0 : TP;
	xMsg2955 : Msg; (* B2955 -  instance of AmBase Library function Msg*)
	xMsg2954 : Msg; (* B2954 -  instance of AmBase Library function Msg*)
	xMsg2953 : Msg; (* B2953 -  instance of AmBase Library function Msg*)
	xMsg2952 : Msg; (* B2952 -  instance of AmBase Library function Msg*)
	xMsg2951 : Msg; (* B2951 -  instance of AmBase Library function Msg*)
	xMsg2950 : Msg; (* B2950 -  instance of AmBase Library function Msg*)
	xMsg2949 : Msg; (* B2949 -  instance of AmBase Library function Msg*)
	xMsg2948 : Msg; (* B2948 -  instance of AmBase Library function Msg*)
	xMsg2947 : Msg; (* B2947 -  instance of AmBase Library function Msg*)
	xMsg2946 : Msg; (* B2946 -  instance of AmBase Library function Msg*)
	xMsg2945 : Msg; (* B2945 -  instance of AmBase Library function Msg*)
	xMsg2944 : Msg; (* B2944 -  instance of AmBase Library function Msg*)
	xMsg2943 : Msg; (* B2943 -  instance of AmBase Library function Msg*)
	xMsg2942 : Msg; (* B2942 -  instance of AmBase Library function Msg*)
	xMsg2941 : Msg; (* B2941 -  instance of AmBase Library function Msg*)
	xMsg2940 : Msg; (* B2940 -  instance of AmBase Library function Msg*)
	xMsg9008 : Msg; (* B9008 -  instance of AmBase Library function Msg*)
	xMsg9009 : Msg; (* B9009 -  instance of AmBase Library function Msg*)
	xMsg9010 : Msg; (* B9010 -  instance of AmBase Library function Msg*)
	xMsg9011 : Msg; (* B9011 -  instance of AmBase Library function Msg*)
	xMsg9012 : Msg; (* B9012 -  instance of AmBase Library function Msg*)
	xMsg9013 : Msg; (* B9013 -  instance of AmBase Library function Msg*)
	xMsg9014 : Msg; (* B9014 -  instance of AmBase Library function Msg*)
	xMsg9015 : Msg; (* B9015 -  instance of AmBase Library function Msg*)
	xMsg9016 : Msg; (* B9016 -  instance of AmBase Library function Msg*)
	xMsg9017 : Msg; (* B9017 -  instance of AmBase Library function Msg*)
	xMsg9018 : Msg; (* B9018 -  instance of AmBase Library function Msg*)
	xMsg9019 : Msg; (* B9019 -  instance of AmBase Library function Msg*)
	xMsg9020 : Msg; (* B9020 -  instance of AmBase Library function Msg*)
	xMsg9021 : Msg; (* B9021 -  instance of AmBase Library function Msg*)
	xMsg9022 : Msg; (* B9022 -  instance of AmBase Library function Msg*)
	xMsg9023 : Msg; (* B9023 -  instance of AmBase Library function Msg*)
	xMsg9093 : Msg; (* B9093 -  instance of AmBase Library function Msg*)
	xMsg9094 : Msg; (* B9094 -  instance of AmBase Library function Msg*)
	xMsg2344 : Msg;
	xMsg2345 : Msg;
END_VAR
```

### Program Logical/Grid/VisGR (IEC, version 4.11.0) - visualization

#### VisGRCyclic.st - Cyclic code
```iecst
(*******************************************************************************
Visualisation grid

This code is confidential AND proprietary TO the INNIO Company.
It may NOT be used in any form, or reproduced in any manner,
without the express written permission OF the INNIO Company.
Copyright, INNIO Company, 2022

Customized modifications: -
------------------------

History:
-------
V4.10.0	16.11.2020  lettenb.	from msy to adapt for +A
V4.11.0 17.01.2022	lettenb.	MM2VIS.bDI_Dem_EU_Block: IN_GR.bEng_Block_EVU added, bugfix

Instructions FOR use:
--------------------
Outstandings:
------------
*******************************************************************************)
PROGRAM _CYCLIC

//MM2VIS.bTestGR 						:= OUT_GR.bTestGR;

MM2VIS.bDI_Dem_EU_Block				:= IN_GR.tDI_Dem_EU_Block.Di OR IN_GR.bEng_Block_EVU;
MM2VIS.bDI_Dem_EU_MnsConBlock;(*	:= IN_GR.tDI_Dem_EU_MnsConBlock.Di; 	(* for future - lock mains connection   1=locked *)
MM2VIS.bLockPlantBC_SetEUCOn; (* 	:= IN_GR.bLockPlantBC_SetEUCOn; 		(* for future - lock plant(all modules) 1=locked *)
MM2VIS.bLockMnsConBC_SetEUCOn;(*	:= IN_GR.bLockMnsConBC_SetEUCOn; 		(* for future - lock mains connection   1=locked *)

MM2VIS.bP_GenC_SetEUCOn				:= IN_GR.bP_GenC_SetEUCOn;
MM2VIS.bP_GenC_SetEUCOf				:= IN_GR.bP_GenC_SetEUCOf;
MM2VIS.rGCP_P;
MM2VIS.bGenC_PBC_SetCOn				:= IN_GR.bGenC_PBC_SetCOn;
MM2VIS.bGenC_PBC_SetCOf				:= IN_GR.bGenC_PBC_SetCOf;
MM2VIS.rGenC_PBC					:= IN_GR.rGenC_PBC;

MM2VIS.bPF_GenC_SetEUCOn			:= IN_GR.bPF_GenC_SetEUCOn;
MM2VIS.bPF_GenC_SetEUCOf 			:= IN_GR.bPF_GenC_SetEUCOf;
MM2VIS.rGCQ_PF;
MM2VIS.bGenC_PFBC_SetCOn			:= IN_GR.bGenC_PFBC_SetCOn;
MM2VIS.bGenC_PFBC_SetCOf			:= IN_GR.bGenC_PFBC_SetCOf;
MM2VIS.rGenC_PFBC					:= IN_GR.rGenC_PFBC;

MM2VIS.bQ_GenC_SetEUCOn				:= IN_GR.bQ_GenC_SetEUCOn;
MM2VIS.bQ_GenC_SetEUCOf 			:= IN_GR.bQ_GenC_SetEUCOf;
MM2VIS.rGCQ_Q;
MM2VIS.bGenC_QBC_SetCOn				:= IN_GR.bGenC_QBC_SetCOn;
MM2VIS.bGenC_QBC_SetCOf				:= IN_GR.bGenC_QBC_SetCOf;
MM2VIS.rGenC_QBC					:= IN_GR.rGenC_QBC;

MM2VIS.bU_GenC_SetEUCOn				:= IN_GR.bU_GenC_SetEUCOn;
MM2VIS.bU_GenC_SetEUCOf				:= IN_GR.bU_GenC_SetEUCOf;
MM2VIS.rGCQ_USet;
MM2VIS.bGenC_UBC_SetCOn				:= IN_GR.bGenC_UBC_SetCOn;
MM2VIS.bGenC_UBC_SetCOf				:= IN_GR.bGenC_UBC_SetCOf;
MM2VIS.rGenC_UQBC					:= IN_GR.rGenC_UQBC;

MM2VIS.bPLim_GenC_SetEUCOn			:= IN_GR.bPLim_GenC_SetEUCOn;
MM2VIS.bPLim_GenC_SetEUCOf			:= IN_GR.bPLim_GenC_SetEUCOf;
MM2VIS.rGCP_PLim_AI;
MM2VIS.bGenC_PLimBC_SetCOn			:= IN_GR.bGenC_PLimBC_SetCOn;
MM2VIS.bGenC_PLimBC_SetCOf			:= IN_GR.bGenC_PLimBC_SetCOf;
MM2VIS.rGenC_PLimBC					:= IN_GR.rGenC_PLimBC;

MM2VIS.bQLim_GenC_SetEUCOn			:= IN_GR.bQLim_GenC_SetEUCOn;
MM2VIS.bQLim_GenC_SetEUCOf			:= IN_GR.bQLim_GenC_SetEUCOf;
MM2VIS.rGCQ_QLim_AI;
MM2VIS.bGenC_QLimBC_SetCOn			:= IN_GR.bGenC_QLimBC_SetCOn;
MM2VIS.bGenC_QLimBC_SetCOf			:= IN_GR.bGenC_QLimBC_SetCOf;
MM2VIS.rGenC_QLimBC;

//MM2VIS.bLFSMO_SetEUCOn				:= IN_GR.bLFSMO_SetEUCOn;	(*TF 3.2.3, plant category C*)
//MM2VIS.bLFSMO_SetEUCOf				:= IN_GR.bLFSMO_SetEUCOf;
//MM2VIS.bLFSMU_SetEUCOn				:= IN_GR.bLFSMU_SetEUCOn;
//MM2VIS.bLFSMU_SetEUCOf				:= IN_GR.bLFSMU_SetEUCOf;
//MM2VIS.bLFSMO_SetEUCOn_BC			:= IN_GR.bLFSMO_SetEUCOn_BC;
//MM2VIS.bLFSMO_SetEUCOf_BC			:= IN_GR.bLFSMO_SetEUCOf_BC;
//MM2VIS.bLFSMU_SetEUCOn_BC			:= IN_GR.bLFSMU_SetEUCOn_BC;
//MM2VIS.bLFSMU_SetEUCOf_BC			:= IN_GR.bLFSMU_SetEUCOf_BC;

MM2VIS.bPRampExt_SetEUCOn			:= IN_GR.tCU2GR.bFSM_Rmp_AI_COn;
MM2VIS.bPRampExtBC_SetEUCOn			:= IN_GR.tCU2GR.bFSM_Rmp_BC_COn;
MM2VIS.rPRampExtBC_SetEU_Up			:= IN_GR.tCU2GR.rP_FSM_Rmp_Up_BC;
MM2VIS.rPRampExtAi_SetEU_Up			:= IN_GR.tHA2GR.tFSM_Rmp_Up.Ai;
MM2VIS.rPRampExtBC_SetEU_Down		:= IN_GR.tCU2GR.rP_FSM_Rmp_Down_BC;
MM2VIS.rPRampExtAi_SetEU_Down		:= IN_GR.tHA2GR.tFSM_Rmp_Down.Ai;

MM2VIS.rU_droopBC					:= IN_GR.tCU2GR.rU_Droop_BC;
MM2VIS.rU_droopAI					:= IN_GR.tHA2GR.tU_Droop.Ai;

MM2VIS.rF_FC_Deadband_posBC			:= IN_GR.tCU2GR.rF_FSMO_DB_BC;
MM2VIS.rF_FC_Deadband_posAi			:= IN_GR.tHA2GR.tF_FSMO_DB.Ai;
MM2VIS.rDroop_FC_posBC				:= IN_GR.tCU2GR.rP_FSMO_Droop_BC;
MM2VIS.rDroop_FC_posAi				:= IN_GR.tHA2GR.tF_FSMO_Droop.Ai;
MM2VIS.rF_FC_Deadband_negBC			:= IN_GR.tCU2GR.rF_FSMU_DB_BC;
MM2VIS.rF_FC_Deadband_negAi			:= IN_GR.tHA2GR.tF_FSMU_DB.Ai;
MM2VIS.rDroop_FC_negBC				:= IN_GR.tCU2GR.rP_FSMU_Droop_BC;
MM2VIS.rDroop_FC_negAi				:= IN_GR.tHA2GR.tF_FSMU_Droop.Ai;

MM2VIS.rF_LFSMU_GrC_DeadBand_negBC	:= IN_GR.tCU2GR.rF_LFSMU_DB_BC;
MM2VIS.rF_LFSMU_GrC_DeadBand_negAi	:= IN_GR.tHA2GR.tF_LFSMU_DB.Ai;
MM2VIS.rDroop_GrC_LFSMU_negBC		:= IN_GR.tCU2GR.rP_LFSMU_Droop_BC;
MM2VIS.rDroop_GrC_LFSMU_negAi		:= IN_GR.tHA2GR.tF_LFSMU_Droop.Ai;
MM2VIS.rF_LFSMO_GrC_DeadBand_posBC	:= IN_GR.tCU2GR.rF_LFSMO_DB_BC;
MM2VIS.rF_LFSMO_GrC_DeadBand_posAi	:= IN_GR.tHA2GR.tF_LFSMO_DB.Ai;
MM2VIS.rDroop_GrC_LFSMO_posBC		:= IN_GR.tCU2GR.rP_LFSMO_Droop_BC;
MM2VIS.rDroop_GrC_LFSMO_posAi		:= IN_GR.tHA2GR.tF_LFSMO_Droop.Ai;

MM2VIS.bFC_SetCOn					:= IN_GR.bFC_SetCOn;
MM2VIS.bFC_SetCOf					:= IN_GR.bFC_SetCOf;
MM2VIS.bSet_FC_COn_Bus				:= IN_GR.bSet_FC_COn_Bus;
MM2VIS.bSet_FC_COf_Bus				:= IN_GR.bSet_FC_COf_Bus;

MM2VIS.bILF_SetCOn					:= IN_GR.bILF_SetCOn;
MM2VIS.bILF_SetCOf					:= IN_GR.bILF_SetCOf;
MM2VIS.bSet_ILF_COn_Bus				:= IN_GR.bSet_ILF_COn_Bus;
MM2VIS.bSet_ILF_COf_Bus				:= IN_GR.bSet_ILF_COf_Bus;

//MM2VIS.rQmns_pv_1					:= IN_GR.tQ_Act[1].Ai;
//MM2VIS.rQmns_sp_1					:= MM2VIS.rQ_set * Para.rS_Nom * (-1);(* change sign for VZS*)
//MM2VIS.rUmns_pv_1					:= IN_GR.tU_Avg[1].Ai;
//MM2VIS.rUmns_sp_1					:= MM2VIS.rU_set * Para.rU_GrC_SetEU_Nom;
//MM2VIS.rPFmns_pv_1					:= IN_GR.tPF_Act[1].Ai;
//MM2VIS.rPFmns_sp_1					:= rPF_EU;

END_PROGRAM
```

#### VisGRInit.st - Initialization code
```iecst
PROGRAM _INIT

(* TODO : Add your code here *)

END_PROGRAM
```

### Package Logical/Gastrain - GT: Gas Train

### Data object Logical/Gastrain/META_GT (Simple) - MODUL META data file

#### META_GT.dat
```
; *******************************************************************************
; AGGR: Module Meta Data (data module)
;
; This code is confidential and proprietary to the INNIO Company.
; It may not be used in any form, or reproduced in any manner, without the express
; written permission of the INNIO Company.
; Copyright, INNIO Company, 2025
;
; Customized modifications: -
; ------------------------
;
; History:
; -------
; V03.99.00.00	06.03.2013	Weitzer		generated for modular software
; V03.99.02.00	29.05.2013	Zengerer	initial dependencies prepared
; V04.00.00.00	30.01.2014	Denk		new version
; V04.00.01.00  24.03.2014	Ze/De	 	VIS OPC Interface change-> VIS dependency added
; V04.00.02.00	20.06.2014	Denk		new version
; V04.01.00.00	22.07.2014	Denk		Para task update, gas counter, MSS(CH4,GD,SD)
; V04.01.01.00 	07.10.2014	Denk		Adicom Pre-chamber gas compressor logic added
; V04.01.02.00 	14.10.2014	Denk		Bugfix O2 max activation
; V04.03.00.00 	08.01.2014	Denk		Porting J920 for XT4 and Bugfix
; V04.03.01.00	02.11.2015	Zengerer 	MANDATORYMODULE statement, version + dependencies changed (IF change with array index 0 for compatibility with c-tasks)
; V04.05.00.00  21.01.2017  Denk		SWAT releases 1,2,3,4. Power reduction gas pressure min.
; V04.05.01.00	24.10.2017	Zingerle	Reduction with difference pressure minimum, implemented
; V04.05.02.00	01.03.2018	Denk		Reduction with difference pressure minimum, Spec. change and validation changes
; V04.05.03.00	23.03.2018	Denk		main gas differential pressure power reduction 1 and 2, limit value: moved to PermGT2
; V04.05.04.00	29.03.2018	Denk		PermGT2, spare values added
; V04.06.00.00	20.09.2018	Perktold	interfaces and functions for fast start added
; V04.07.00.00	30.04.2018	Denk	 	SWAT Rel.5, change A2289 to W2570
;										SWAT Rel.5, W3445 delay time
;										SWAT Rel.5, A1095 deleted for type9
;										SWAT Rel.5, A1085 delay time for type 9 changed to 3s
;										SWAT Rel.5, deactivation of A3376 when pressure based control is active
;				04.07.2018	Denk		Bugfix, Anzeige Leistungsreduktion Gasdruck min.
;				24.09.2018	Denk		Avoid second start of gas safety device (DPFR-20180821-0202)
;				05.02.2019	Denk		Bugfix, PermGT and PermGT2: ModulName STRING[9] changed to STRING[35]
;				15.02.2019	Denk		Bugfix, when parameter 11363 is TRUE, AutGas was not active after PLC warmstart.
; V04.07.00.00	22.03.2019	Zengerer 	Several new features and TKE customisation variants implemented from Spec Gastrain Requisition 2018
; V04.09.00.00	5.6.-16.1.2020	Zengerr iGasTrain_Type, tiGT_TestDuration
; 				27.06.2019	Denk		Additional measurements in natural gas train
; V04.10.00.00	05.08.2020  Zuschnig	Added control of dome blow off valve
;				08.12.2020	Denk		Bugfix, xTON_GDMA2() changed to xTON_GDMA2_VISA()
;       	    10.12.2020  Zuschnig	Included power reduction for Tecjet differential pressure
;				21.01.2021  Zuschnig	Bugfix, Power reduction suction pressure (swap X1<->X2)
;				28.01.2021	Denk		Alarm deactivation when DGS/WinMOD Simulation is active (2261, 3376, 3377, 3444, 3445).
; V04.11.00.00	22.06.2021	Arnold		J6 data center application
;				21.10.2021	Zuschnig	Update prechamber gas train power reduction
;				20.01.2022  Zuschnig	Update gas rail pressure power reduction
;				28.01.2022	Perktold	included plant controller upgrade
;				11.02.2022	Zuschnig	Remove engine demand for release of upstream gas valve
;				02.03.2022	Zuschnig	Include CH4 signal via Bus from customize modul
;				17.03.2022	Zuschnig	Use standard label from customized modul for gasmixing setpoint
;               18.03.2022  Zuschnig    Rework of gas counter impulse prescaler
;				18.03.2022	Zuschnig	Removed fixed spare parameter and customized analog input
; V04.12.00.00	23.08.2022	Zuschnig	Initialize standard value for power redcution gas rail pressure
;				07.11.2022	Zuschnig	Include gas pressure min/max from customized module for gas train 1
;				22.01.2023	Zuschnig	Include H2 measurement
; V04.13.00.00  20.06.2023  Zuschnig	Added standardized AI input for gas mixing ratio
;				30.11.2023	Goenczi		puffmini hold gas valve for GCB opening by Customer control
;				05.12.2023	Zuschnig	Update prechamber gas train power reduction in island mode
;				06.12.2023	Zuschnig	Replace IN_GT.bSA_PI_Active with Para.bSA_PI_Active
;				28.02.2024	Zuschnig	Include Para.bGCActive for setting A3326
; V04.14.00.00  09.07.2024  Schmidt		T6L version during load acceptance: reduce limit difference pressure prechamber minimum
;				06.11.2024	Kafka		fast gastrain for Gen2 T9
;				22.11.2024	Schmidt		Added pre chamber gas bypass valve logic (load acceptance improvements)
;				28.11.2024	Nagy		Modified A1084, A1085, A3003 - 2024-222 GasTrain Desensitization
;				11.12.2024	Zuschnig	Prechamber gas train power reduction in island mode - W9387 only if reduced power < 1
;				23.02.2025	Tinello		Gas leakage check moved to SafetyPLC
; V04.25.00.00	30.12.2025	Tinello		Logic modified because of SafetyPLC
;
; Instructions for use:
; --------------------
; make only changes at the version numbers
; OBEY XML FORMATING RULES!
;
; Outstandings:
; ------------
;CHECK tiGT_TestDuration' MIN='1' MAX='120'
; *******************************************************************************
;
"<META>"
;
; Module ID
"<MODUL>GT</MODUL>"
;
; Module Version (xx.yy.zz.cc)
"<VERSION>04.25.00.00</VERSION>"
;
; Module Basisupdate Version BU (00-99)
"<BASISUPDATE_VERSION>00</BASISUPDATE_VERSION>"
;
; Optional: specify order number for limitated module usage
"<ORDER></ORDER>" ;<!--(optional for restricted customizations; missing statement makes module valid for all orders)-->
;
; Parameter Check <PARAn Name='aAbcdef' MIN='xxx' MAX='yyy' />  (watch for correct spacings and apostrophs!)
"<PARAMETER_CHK>"
"	<PARA1 Name='rN_EngStart_LimHi' MIN='50.0' MAX='2200.0' />"
"	<PARA2 Name='iEng_Motortype ' MIN='208' MAX='920' />"
"	<PARA3 Name='iGasTrain_Type' MIN='1' MAX='4' />"
"	<PARA4 />"
"	<PARA5 />"
"</PARAMETER_CHK>"
;
; Statement, if engine operation is also allowed without this module (FALSE) or if this module´s parameter check passing is mandatory (TRUE)
"<MANDATORYMODULE>TRUE</MANDATORYMODULE>"
;
; Permanent Datamodule Filenames<!-- NAME ist ohne Dateiendung einzutragen; Nur für Counter und interne Parameter verwenden-->
"<DATAMODULES>" ;<!-- optional; mehrere DATAMODULES erlaubt-->
"	<DATAMODULE>par_GT</DATAMODULE>"
"	<DATAMODULE>perm_GT</DATAMODULE>"
"	<DATAMODULE>perm_GT2</DATAMODULE>"
"</DATAMODULES>"
;
; Dependencies Modules (MMxx.yy.zz.cc)
"<DEPENDENCIES>"
"	<DEPENDENCY MODULE='AB' VERSION='04.00.00.00' />"
"	<DEPENDENCY MODULE='AG' VERSION='04.00.00.00' />"
"	<DEPENDENCY MODULE='CU' VERSION='04.07.02.00' />"
"	<DEPENDENCY MODULE='EC' VERSION='04.14.00.00' />"
"	<DEPENDENCY MODULE='EG' VERSION='04.25.00.00' />"
"	<DEPENDENCY MODULE='EX' VERSION='04.00.00.00' />"
"	<DEPENDENCY MODULE='HA' VERSION='04.14.00.00' />"
"	<DEPENDENCY MODULE='IG' VERSION='04.00.00.00' />"
"	<DEPENDENCY MODULE='OP' VERSION='04.13.00.00' />"
"	<DEPENDENCY MODULE='SY' VERSION='04.04.00.00' />"
"	<DEPENDENCY MODULE='PB' VERSION='04.00.00.00' />"
"	<DEPENDENCY MODULE='CH' VERSION='04.04.00.00' />"
"	<DEPENDENCY MODULE='GD' VERSION='04.10.00.00' />"
"	<DEPENDENCY VISVERSION='02.15.00.00' />" 			;Dependencies Visualization
"</DEPENDENCIES>"
;
; Module function description
"<MODULEFUNCTION>" ;<!-- short overview documentation of module function; add reference to detailed information, if available-->
"	<General>	"
"	 Control and monitoring Gastrain	"
"	</General>	"
""
"	<F1 Name='Special gas' LastModified='04.00.00.00'>"
"	 Monitoring and control of special gas engines (messages, power reduction).	"
"	</F1>"
"	<F2 Name='Biogas' LastModified='04.00.00.00'>"
"	 Control and monitoring gas blower/flare.	"
"	</F2>"
"	<F3 Name='Gastrain and prechamber gas train' LastModified='04.00.00.00'>"
"	 Control gastrain and prechamber gastrain regarding pressure limits.  "
"	</F3>"
"	<F4 Name='Gas mixing' LastModified='04.00.00.00'>"
"	 Control gas mixing with flaps/valves or Tecjet.  "
"	</F4>"
"	<F5 Name='Data calculation' LastModified='04.00.00.00'>"
"	 Calculaltion of operation/normal cubic meter and gas volume correction factor.	"
"	</F5>"
"	<F6 Name='Gastrain testing' LastModified='04.00.00.00'>"
"	 Testing Gastrain 1 and 2 (Leak tightness).	"
"	</F6>"
"	<F7 Name='Gas valves' LastModified='04.00.00.00'>"
"	 Control and release gas valves.	"
"	</F7>"
"	<F8 Name='Pre-chamber gas compressor' LastModified='04.00.00.00'>"
"	 Control Pre-chamber gas compressor.	"
"	</F8>"
"	<F9 Name='Deflagration protection' LastModified='04.00.00.00'>"
"	 Deflagration protection for engine type 6 and 9.	"
"	</F9>"
""
"	<Info>"
"	 V04.01.00	Gas counter parameters added 	"
"	 V04.03.00	J920 functionalities added 	"
" 	 V04.05.00	Serienvorbereitung Gasmischung mit tCustAnaIn[1] oder IN_GT.rGT_RatioMix_Set "
"    V04.05.00	version + dependencies changed (IF change with array index 0 for compatibility with c-tasks)	"
"    V04.05.00  SWAT Desensitization changes for type9	"
"    V04.07.00  TKE customisation variants integrated	"
"    V04.09.00  Additional Measurements in natural gas train, META Gas Valve handling	"
"	</Info>"
""
"	<Customized LastModified='4.07.0.0'>	"
"	- Nothing "
"	</Customized>	"
""
"</MODULEFUNCTION>"
;
"</META>"
```
